C05453=1097.627,129.752,-63.111,176.753,16.480,152.163
C05454=1097.633,130.001,-63.131,176.756,16.481,152.163
C05455=1097.638,130.250,-63.150,176.760,16.481,152.162
C05456=1097.644,130.499,-63.171,176.762,16.481,152.162
C05457=1097.649,130.749,-63.190,176.765,16.482,152.161
C05458=1097.656,130.998,-63.210,176.768,16.482,152.161
C05459=1097.661,131.248,-63.229,176.771,16.482,152.160
C05460=1097.667,131.496,-63.249,176.774,16.482,152.159
C05461=1097.673,131.745,-63.270,176.777,16.482,152.159
C05462=1097.678,131.995,-63.289,176.780,16.482,152.158
C05463=1097.684,132.244,-63.309,176.783,16.483,152.158
C05464=1097.690,132.493,-63.329,176.785,16.483,152.157
C05465=1097.695,132.742,-63.349,176.789,16.483,152.157
C05466=1097.701,132.991,-63.369,176.792,16.484,152.156
C05467=1097.706,133.241,-63.389,176.794,16.484,152.156
C05468=1097.712,133.490,-63.409,176.798,16.484,152.155
C05469=1097.718,133.738,-63.429,176.801,16.484,152.155
C05470=1097.724,133.988,-63.449,176.803,16.485,152.154
C05471=1097.729,134.237,-63.468,176.806,16.485,152.154
C05472=1097.734,134.486,-63.489,176.810,16.485,152.153
C05473=1097.740,134.735,-63.509,176.812,16.485,152.152
C05474=1097.746,134.984,-63.528,176.815,16.485,152.152
C05475=1097.751,135.234,-63.549,176.819,16.486,152.151
C05476=1097.757,135.482,-63.569,176.821,16.486,152.151
C05477=1097.763,135.731,-63.589,176.824,16.486,152.150
C05478=1097.768,135.981,-63.608,176.828,16.486,152.150
C05479=1097.774,136.230,-63.629,176.830,16.486,152.149
C05480=1097.780,136.479,-63.649,176.833,16.487,152.149
C05481=1097.786,136.728,-63.669,176.836,16.487,152.148
C05482=1097.791,136.977,-63.689,176.839,16.487,152.147
C05483=1097.797,137.226,-63.709,176.842,16.488,152.147
C05484=1097.802,137.475,-63.729,176.845,16.488,152.146
C05485=1097.808,137.724,-63.749,176.848,16.488,152.146
C05486=1097.814,137.974,-63.770,176.851,16.488,152.145
C05487=1097.820,138.223,-63.790,176.854,16.489,152.145
C05488=1097.825,138.472,-63.811,176.857,16.488,152.144
C05489=1097.831,138.721,-63.831,176.860,16.489,152.143
C05490=1097.836,138.970,-63.850,176.863,16.489,152.143
C05491=1097.842,139.219,-63.870,176.866,16.489,152.142
C05492=1097.847,139.468,-63.891,176.869,16.489,152.142
C05493=1097.853,139.717,-63.911,176.872,16.490,152.141
C05494=1097.858,139.966,-63.931,176.875,16.489,152.141
C05495=1097.864,140.216,-63.952,176.878,16.490,152.140
C05496=1097.870,140.465,-63.972,176.881,16.490,152.139
C05497=1097.875,140.714,-63.993,176.884,16.490,152.139
C05498=1097.881,140.963,-64.013,176.887,16.490,152.138
C05499=1097.887,141.212,-64.033,176.890,16.490,152.138
C05500=1097.892,141.461,-64.054,176.893,16.490,152.137
C05501=1097.898,141.710,-64.074,176.896,16.491,152.137
C05502=1097.903,141.959,-64.094,176.899,16.491,152.136
C05503=1097.909,142.209,-64.115,176.902,16.491,152.135
C05504=1097.915,142.458,-64.135,176.905,16.491,152.135
C05505=1097.920,142.707,-64.156,176.908,16.492,152.134
C05506=1097.926,142.956,-64.176,176.912,16.492,152.134
C05507=1097.932,143.205,-64.196,176.914,16.492,152.133
C05508=1097.937,143.454,-64.217,176.917,16.492,152.133
C05509=1097.944,143.729,-64.240,176.921,16.492,152.132
C05510=1097.950,144.003,-64.262,176.924,16.492,152.131
C05511=1097.956,144.278,-64.286,176.928,16.492,152.130
C05512=1097.962,144.552,-64.308,176.931,16.493,152.130
C05513=1097.967,144.801,-64.329,176.934,16.493,152.129
C05514=1097.973,145.050,-64.348,176.937,16.493,152.129
C05515=1097.979,145.300,-64.369,176.940,16.493,152.128
C05516=1097.985,145.549,-64.390,176.943,16.493,152.128
C05517=1097.990,145.798,-64.410,176.946,16.493,152.127
C05518=1097.996,146.046,-64.431,176.949,16.493,152.126
C05519=1098.001,146.295,-64.452,176.953,16.494,152.126
C05520=1098.007,146.545,-64.473,176.955,16.493,152.125
C05521=1098.013,146.794,-64.493,176.959,16.494,152.125
C05522=1098.019,147.043,-64.513,176.962,16.494,152.124
C05523=1098.024,147.291,-64.534,176.964,16.494,152.123
C05524=1098.030,147.541,-64.555,176.968,16.494,152.123
C05525=1098.035,147.790,-64.576,176.971,16.494,152.122
C05526=1098.041,148.039,-64.596,176.974,16.494,152.122
C05527=1098.047,148.288,-64.617,176.977,16.494,152.121
C05528=1098.053,148.537,-64.638,176.980,16.494,152.120
C05529=1098.058,148.787,-64.659,176.984,16.495,152.120
C05530=1098.063,149.035,-64.680,176.986,16.494,152.119
C05531=1098.069,149.285,-64.701,176.989,16.495,152.119
C05532=1098.075,149.534,-64.721,176.993,16.495,152.118
C05533=1098.081,149.782,-64.742,176.995,16.495,152.117
C05534=1098.086,150.031,-64.763,176.999,16.495,152.117
C05535=1098.092,150.281,-64.783,177.002,16.495,152.116
C05536=1098.097,150.530,-64.805,177.005,16.495,152.115
C05537=1098.103,150.779,-64.825,177.008,16.495,152.115
C05538=1098.108,151.028,-64.846,177.012,16.495,152.114
C05539=1098.114,151.277,-64.868,177.015,16.496,152.114
C05540=1098.119,151.526,-64.888,177.017,16.495,152.113
C05541=1098.125,151.775,-64.909,177.021,16.496,152.112
C05542=1098.131,152.025,-64.930,177.024,16.496,152.112
C05543=1098.137,152.273,-64.951,177.027,16.495,152.111
C05544=1098.142,152.522,-64.971,177.030,16.495,152.110
C05545=1098.148,152.772,-64.992,177.033,16.496,152.110
C05546=1098.154,153.020,-65.014,177.037,16.496,152.109
C05547=1098.159,153.269,-65.034,177.039,16.496,152.109
C05548=1098.165,153.519,-65.056,177.043,16.496,152.108
C05549=1098.170,153.768,-65.076,177.046,16.496,152.107
C05550=1098.176,154.016,-65.098,177.049,16.496,152.107
C05551=1098.182,154.266,-65.119,177.052,16.496,152.106
C05552=1098.187,154.515,-65.140,177.055,16.496,152.105
C05553=1098.193,154.763,-65.161,177.059,16.496,152.105
C05554=1098.199,155.013,-65.182,177.061,16.496,152.104
C05555=1098.204,155.261,-65.203,177.065,16.496,152.104
C05556=1098.210,155.511,-65.224,177.068,16.497,152.103
C05557=1098.216,155.760,-65.246,177.071,16.496,152.102
C05558=1098.221,156.009,-65.266,177.074,16.496,152.102
C05559=1098.227,156.258,-65.288,177.078,16.496,152.101
C05560=1098.232,156.507,-65.310,177.081,16.497,152.100
C05561=1098.238,156.757,-65.330,177.084,16.496,152.100
C05562=1098.244,157.005,-65.352,177.087,16.497,152.099
C05563=1098.249,157.254,-65.373,177.090,16.496,152.098
C05564=1098.255,157.504,-65.394,177.094,16.497,152.098
C05565=1098.261,157.752,-65.415,177.096,16.496,152.097
C05566=1098.267,158.001,-65.437,177.100,16.497,152.097
C05567=1098.272,158.250,-65.457,177.103,16.497,152.096
C05568=1098.277,158.499,-65.479,177.106,16.496,152.095
C05569=1098.283,158.748,-65.501,177.109,16.496,152.095
C05570=1098.288,158.997,-65.521,177.112,16.497,152.094
C05571=1098.294,159.247,-65.543,177.116,16.497,152.093
C05572=1098.300,159.495,-65.564,177.118,16.497,152.093
C05573=1098.306,159.770,-65.588,177.122,16.497,152.092
C05574=1098.312,160.044,-65.611,177.126,16.496,152.091
C05575=1098.319,160.318,-65.635,177.129,16.496,152.091
C05576=1098.325,160.592,-65.659,177.133,16.496,152.090
C05577=1098.331,160.842,-65.680,177.136,16.496,152.089
C05578=1098.335,161.090,-65.701,177.139,16.497,152.089
C05579=1098.342,161.340,-65.723,177.143,16.497,152.088
C05580=1098.347,161.588,-65.744,177.146,16.497,152.087
C05581=1098.353,161.837,-65.766,177.149,16.496,152.087
C05582=1098.358,162.086,-65.788,177.152,16.497,152.086
C05583=1098.364,162.336,-65.809,177.156,16.497,152.085
C05584=1098.370,162.585,-65.830,177.158,16.497,152.085
C05585=1098.374,162.833,-65.852,177.162,16.497,152.084
C05586=1098.381,163.083,-65.874,177.165,16.497,152.083
C05587=1098.385,163.331,-65.895,177.169,16.497,152.083
C05588=1098.392,163.581,-65.917,177.171,16.496,152.082
C05589=1098.396,163.829,-65.939,177.175,16.497,152.081
C05590=1098.403,164.079,-65.961,177.178,16.497,152.081
C05591=1098.408,164.327,-65.982,177.181,16.497,152.080
C05592=1098.413,164.577,-66.004,177.184,16.497,152.079
C05593=1098.419,164.825,-66.025,177.188,16.497,152.079
C05594=1098.424,165.074,-66.047,177.191,16.497,152.078
C05595=1098.430,165.323,-66.069,177.195,16.497,152.077
C05596=1098.435,165.572,-66.091,177.198,16.497,152.077
C05597=1098.441,165.821,-66.112,177.201,16.497,152.076
C05598=1098.446,166.070,-66.134,177.204,16.497,152.075
C05599=1098.452,166.319,-66.156,177.207,16.497,152.075
C05600=1098.457,166.568,-66.178,177.211,16.497,152.074
C05601=1098.463,166.817,-66.199,177.214,16.496,152.073
C05602=1098.469,167.066,-66.221,177.217,16.497,152.073
C05603=1098.474,167.315,-66.243,177.221,16.497,152.072
C05604=1098.480,167.564,-66.264,177.224,16.497,152.071
C05605=1098.485,167.813,-66.286,177.227,16.497,152.071
C05606=1098.491,168.062,-66.308,177.230,16.497,152.070
C05607=1098.496,168.311,-66.330,177.234,16.497,152.069
C05608=1098.502,168.560,-66.351,177.237,16.497,152.069
C05609=1098.507,168.809,-66.374,177.240,16.496,152.068
C05610=1098.513,169.058,-66.396,177.243,16.496,152.067
C05611=1098.519,169.307,-66.418,177.247,16.496,152.067
C05612=1098.524,169.556,-66.440,177.250,16.497,152.066
C05613=1098.530,169.805,-66.461,177.254,16.497,152.065
C05614=1098.535,170.054,-66.483,177.256,16.496,152.065
C05615=1098.541,170.303,-66.506,177.260,16.496,152.064
C05616=1098.546,170.552,-66.527,177.263,16.496,152.063
C05617=1098.552,170.801,-66.549,177.267,16.496,152.063
C05618=1098.558,171.050,-66.571,177.269,16.496,152.062
C05619=1098.563,171.298,-66.593,177.273,16.496,152.061
C05620=1098.569,171.548,-66.616,177.276,16.496,152.061
C05621=1098.574,171.797,-66.638,177.280,16.496,152.060
C05622=1098.580,172.046,-66.659,177.283,16.496,152.059
C05623=1098.586,172.295,-66.682,177.286,16.495,152.059
C05624=1098.592,172.544,-66.704,177.290,16.495,152.058
C05625=1098.597,172.793,-66.726,177.293,16.495,152.057
C05626=1098.602,173.042,-66.748,177.297,16.495,152.056
C05627=1098.608,173.291,-66.770,177.299,16.495,152.056
C05628=1098.613,173.540,-66.792,177.303,16.495,152.055
C05629=1098.620,173.788,-66.814,177.306,16.495,152.054
C05630=1098.625,174.038,-66.837,177.310,16.495,152.054
C05631=1098.630,174.287,-66.858,177.313,16.495,152.053
C05632=1098.636,174.535,-66.881,177.316,16.495,152.052
C05633=1098.642,174.785,-66.903,177.320,16.495,152.052
C05634=1098.647,175.033,-66.926,177.323,16.494,152.051
C05635=1098.653,175.282,-66.947,177.327,16.494,152.050
C05636=1098.659,175.532,-66.969,177.329,16.494,152.049
C05637=1098.665,175.805,-66.994,177.334,16.494,152.049
C05638=1098.671,176.079,-67.019,177.338,16.494,152.048
C05639=1098.678,176.353,-67.043,177.341,16.494,152.047
C05640=1098.683,176.626,-67.068,177.345,16.493,152.046
C05641=1098.689,176.876,-67.089,177.349,16.493,152.045
C05642=1098.695,177.124,-67.112,177.351,16.493,152.045
C05643=1098.700,177.374,-67.135,177.355,16.493,152.044
C05644=1098.707,177.623,-67.157,177.358,16.493,152.043
C05645=1098.712,177.871,-67.180,177.362,16.493,152.043
C05646=1098.718,178.120,-67.202,177.365,16.492,152.042
C05647=1098.723,178.369,-67.225,177.368,16.492,152.041
C05648=1098.729,178.618,-67.246,177.372,16.492,152.040
C05649=1098.735,178.867,-67.269,177.375,16.492,152.040
C05650=1098.740,179.116,-67.291,177.379,16.492,152.039
C05651=1098.746,179.365,-67.314,177.382,16.491,152.038
C05652=1098.752,179.614,-67.336,177.385,16.491,152.038
C05653=1098.758,179.863,-67.359,177.389,16.491,152.037
C05654=1098.763,180.112,-67.382,177.392,16.491,152.036
C05655=1098.770,180.361,-67.404,177.396,16.491,152.035
C05656=1098.775,180.609,-67.426,177.399,16.490,152.035
C05657=1098.780,180.858,-67.449,177.402,16.490,152.034
C05658=1098.786,181.107,-67.472,177.406,16.490,152.033
C05659=1098.792,181.356,-67.493,177.410,16.490,152.032
C05660=1098.798,181.605,-67.516,177.413,16.490,152.032
C05661=1098.804,181.854,-67.539,177.416,16.490,152.031
C05662=1098.809,182.103,-67.562,177.420,16.489,152.030
C05663=1098.814,182.352,-67.584,177.423,16.489,152.029
C05664=1098.821,182.600,-67.606,177.427,16.489,152.029
C05665=1098.826,182.849,-67.629,177.430,16.489,152.028
C05666=1098.832,183.098,-67.652,177.433,16.489,152.027
C05667=1098.838,183.348,-67.675,177.437,16.488,152.026
C05668=1098.843,183.597,-67.698,177.440,16.488,152.026
C05669=1098.850,183.845,-67.720,177.444,16.488,152.025
C05670=1098.856,184.094,-67.743,177.448,16.488,152.024
C05671=1098.861,184.343,-67.766,177.451,16.487,152.023
C05672=1098.867,184.592,-67.789,177.454,16.487,152.023
C05673=1098.872,184.841,-67.811,177.458,16.487,152.022
C05674=1098.878,185.090,-67.834,177.461,16.487,152.021
C05675=1098.884,185.339,-67.857,177.465,16.487,152.020
C05676=1098.889,185.587,-67.879,177.469,16.487,152.020
C05677=1098.895,185.836,-67.902,177.471,16.486,152.019
C05678=1098.900,186.085,-67.925,177.475,16.486,152.018
C05679=1098.906,186.334,-67.948,177.478,16.486,152.017
C05680=1098.912,186.583,-67.971,177.482,16.486,152.017
C05681=1098.918,186.832,-67.994,177.486,16.486,152.016
C05682=1098.923,187.081,-68.017,177.489,16.486,152.015
C05683=1098.927,187.330,-68.040,177.492,16.485,152.015
C05684=1098.933,187.579,-68.062,177.496,16.485,152.014
C05685=1098.939,187.828,-68.085,177.499,16.485,152.013
C05686=1098.945,188.077,-68.108,177.503,16.485,152.012
C05687=1098.950,188.326,-68.131,177.506,16.485,152.012
C05688=1098.956,188.574,-68.154,177.510,16.485,152.011
C05689=1098.961,188.824,-68.178,177.513,16.484,152.010
C05690=1098.967,189.073,-68.201,177.516,16.484,152.009
C05691=1098.973,189.321,-68.224,177.520,16.484,152.009
C05692=1098.979,189.570,-68.247,177.523,16.484,152.008
C05693=1098.984,189.818,-68.270,177.527,16.484,152.007
C05694=1098.989,190.067,-68.293,177.531,16.483,152.006
C05695=1098.994,190.316,-68.316,177.534,16.483,152.006
C05696=1099.000,190.565,-68.339,177.537,16.483,152.005
C05697=1099.006,190.814,-68.362,177.541,16.483,152.004
C05698=1099.012,191.063,-68.385,177.545,16.482,152.003
C05699=1099.017,191.312,-68.409,177.548,16.482,152.003
C05700=1099.022,191.561,-68.432,177.552,16.482,152.002
C05701=1099.029,191.834,-68.458,177.555,16.482,152.001
C05702=1099.035,192.108,-68.483,177.559,16.482,152.000
C05703=1099.041,192.381,-68.509,177.563,16.482,151.999
C05704=1099.047,192.654,-68.535,177.567,16.481,151.998
C05705=1099.053,192.903,-68.557,177.570,16.481,151.998
C05706=1099.059,193.152,-68.580,177.574,16.481,151.997
C05707=1099.064,193.401,-68.604,177.578,16.481,151.996
C05708=1099.070,193.650,-68.627,177.581,16.481,151.995
C05709=1099.076,193.899,-68.651,177.584,16.480,151.995
C05710=1099.081,194.147,-68.674,177.588,16.480,151.994
C05711=1099.086,194.397,-68.697,177.591,16.480,151.993
C05712=1099.092,194.645,-68.721,177.595,16.479,151.992
C05713=1099.098,194.894,-68.744,177.599,16.479,151.992
C05714=1099.103,195.143,-68.767,177.602,16.479,151.991
C05715=1099.109,195.391,-68.791,177.606,16.479,151.990
C05716=1099.115,195.641,-68.814,177.609,16.478,151.989
C05717=1099.120,195.890,-68.838,177.613,16.478,151.988
C05718=1099.126,196.138,-68.861,177.616,16.478,151.988
C05719=1099.132,196.387,-68.884,177.620,16.478,151.987
C05720=1099.137,196.637,-68.908,177.623,16.477,151.986
C05721=1099.143,196.885,-68.932,177.627,16.478,151.985
C05722=1099.149,197.134,-68.954,177.631,16.477,151.984
C05723=1099.154,197.382,-68.979,177.634,16.477,151.984
C05724=1099.160,197.631,-69.002,177.637,16.476,151.983
C05725=1099.166,197.881,-69.025,177.641,16.476,151.982
C05726=1099.172,198.129,-69.049,177.645,16.476,151.981
C05727=1099.177,198.378,-69.072,177.648,16.476,151.981
C05728=1099.183,198.627,-69.096,177.652,16.475,151.980
C05729=1099.188,198.876,-69.119,177.656,16.475,151.979
C05730=1099.194,199.124,-69.143,177.660,16.475,151.978
C05731=1099.199,199.373,-69.167,177.662,16.474,151.977
C05732=1099.206,199.622,-69.191,177.666,16.474,151.977
C05733=1099.212,199.871,-69.214,177.670,16.474,151.976
C05734=1099.217,200.120,-69.238,177.674,16.473,151.975
C05735=1099.223,200.368,-69.261,177.677,16.473,151.974
C05736=1099.228,200.617,-69.285,177.681,16.473,151.973
C05737=1099.235,200.866,-69.309,177.684,16.473,151.973
C05738=1099.240,201.115,-69.332,177.688,16.473,151.972
C05739=1099.246,201.364,-69.356,177.691,16.472,151.971
C05740=1099.252,201.612,-69.380,177.695,16.472,151.970
C05741=1099.257,201.862,-69.404,177.699,16.471,151.969
C05742=1099.263,202.110,-69.427,177.702,16.471,151.969
C05743=1099.269,202.359,-69.452,177.706,16.471,151.968
C05744=1099.274,202.608,-69.475,177.710,16.470,151.967
C05745=1099.280,202.856,-69.499,177.713,16.470,151.966
C05746=1099.286,203.105,-69.523,177.717,16.470,151.965
C05747=1099.291,203.354,-69.547,177.720,16.469,151.965
C05748=1099.297,203.603,-69.570,177.724,16.469,151.964
C05749=1099.303,203.851,-69.594,177.727,16.469,151.963
C05750=1099.308,204.100,-69.618,177.731,16.469,151.962
C05751=1099.314,204.349,-69.642,177.735,16.469,151.962
C05752=1099.320,204.598,-69.666,177.739,16.468,151.961
C05753=1099.325,204.847,-69.691,177.742,16.468,151.960
C05754=1099.331,205.095,-69.713,177.746,16.468,151.959
C05755=1099.337,205.345,-69.738,177.750,16.468,151.958
C05756=1099.342,205.593,-69.762,177.753,16.467,151.957
C05757=1099.348,205.842,-69.786,177.756,16.466,151.957
C05758=1099.353,206.090,-69.810,177.760,16.466,151.956
C05759=1099.359,206.340,-69.834,177.764,16.466,151.955
C05760=1099.365,206.588,-69.858,177.767,16.466,151.954
C05761=1099.370,206.837,-69.882,177.771,16.466,151.953
C05762=1099.375,207.086,-69.906,177.775,16.465,151.953
C05763=1099.382,207.335,-69.930,177.778,16.465,151.952
C05764=1099.387,207.583,-69.955,177.782,16.465,151.951
C05765=1099.410,208.592,-70.052,177.824,16.478,151.946
C05766=1099.419,208.961,-70.089,177.829,16.479,151.945
C05767=1099.427,209.331,-70.125,177.833,16.480,151.944
C05768=1099.436,209.701,-70.161,177.839,16.480,151.943
C05769=1099.444,210.070,-70.197,177.844,16.482,151.942
C05770=1099.450,210.320,-70.222,177.847,16.482,151.941
C05771=1099.455,210.568,-70.246,177.851,16.482,151.941
C05772=1099.461,210.818,-70.271,177.855,16.483,151.940
C05773=1099.466,211.066,-70.296,177.858,16.484,151.940
C05774=1099.472,211.314,-70.320,177.861,16.484,151.939
C05775=1099.478,211.563,-70.344,177.864,16.485,151.939
C05776=1099.483,211.812,-70.369,177.868,16.485,151.938
C05777=1099.489,212.061,-70.393,177.872,16.486,151.938
C05778=1099.494,212.309,-70.418,177.875,16.486,151.937
C05779=1099.500,212.558,-70.443,177.878,16.487,151.936
C05780=1099.506,212.807,-70.467,177.882,16.487,151.936
C05781=1099.511,213.056,-70.491,177.885,16.488,151.935
C05782=1099.517,213.304,-70.517,177.889,16.489,151.935
C05783=1099.522,213.553,-70.541,177.892,16.489,151.934
C05784=1099.528,213.802,-70.566,177.895,16.490,151.934
C05785=1099.534,214.051,-70.590,177.899,16.490,151.933
C05786=1099.539,214.299,-70.615,177.903,16.492,151.932
C05787=1099.545,214.548,-70.639,177.906,16.492,151.932
C05788=1099.550,214.797,-70.664,177.909,16.493,151.931
C05789=1099.557,215.045,-70.689,177.912,16.493,151.931
C05790=1099.561,215.294,-70.714,177.916,16.494,151.930
C05791=1099.567,215.543,-70.739,177.920,16.494,151.930
C05792=1099.573,215.792,-70.764,177.923,16.495,151.929
C05793=1099.579,216.041,-70.788,177.926,16.495,151.928
C05794=1099.584,216.289,-70.813,177.930,16.496,151.928
C05795=1099.590,216.538,-70.838,177.934,16.497,151.927
C05796=1099.596,216.786,-70.863,177.937,16.497,151.927
C05797=1099.601,217.036,-70.888,177.940,16.498,151.926
C05798=1099.606,217.284,-70.913,177.943,16.498,151.926
C05799=1099.612,217.533,-70.938,177.947,16.499,151.925
C05800=1099.618,217.782,-70.962,177.951,16.500,151.925
C05801=1099.624,218.030,-70.987,177.954,16.500,151.924
C05802=1099.628,218.279,-71.012,177.957,16.501,151.923
C05803=1099.635,218.528,-71.037,177.961,16.502,151.923
C05804=1099.640,218.776,-71.062,177.965,16.502,151.922
C05805=1099.646,219.025,-71.087,177.968,16.503,151.922
C05806=1099.652,219.273,-71.112,177.971,16.503,151.921
C05807=1099.657,219.523,-71.137,177.975,16.504,151.921
C05808=1099.663,219.771,-71.162,177.978,16.505,151.920
C05809=1099.668,220.020,-71.187,177.982,16.505,151.919
C05810=1099.675,220.269,-71.212,177.985,16.506,151.919
C05811=1099.679,220.517,-71.238,177.989,16.507,151.918
C05812=1099.685,220.766,-71.262,177.992,16.507,151.918
C05813=1099.692,221.015,-71.288,177.995,16.508,151.917
C05814=1099.697,221.263,-71.313,177.999,16.508,151.917
C05815=1099.702,221.512,-71.338,178.003,16.509,151.916
C05816=1099.708,221.760,-71.363,178.006,16.510,151.915
C05817=1099.714,222.009,-71.388,178.009,16.510,151.915
C05818=1099.723,222.383,-71.426,178.014,16.511,151.914
C05819=1099.731,222.757,-71.464,178.020,16.512,151.913
C05820=1099.739,223.131,-71.501,178.025,16.514,151.913
C05821=1099.748,223.504,-71.540,178.030,16.514,151.912
C05822=1099.753,223.753,-71.565,178.033,16.515,151.911
C05823=1099.759,224.001,-71.590,178.037,16.516,151.910
C05824=1099.764,224.250,-71.615,178.041,16.517,151.910
C05825=1099.770,224.498,-71.641,178.044,16.517,151.909
C05826=1099.775,224.747,-71.667,178.047,16.518,151.909
C05827=1099.781,224.995,-71.692,178.051,16.519,151.908
C05828=1099.786,225.245,-71.717,178.054,16.519,151.908
C05829=1099.792,225.494,-71.742,178.058,16.520,151.907
C05830=1099.797,225.742,-71.768,178.062,16.521,151.907
C05831=1099.804,225.991,-71.793,178.065,16.521,151.906
C05832=1099.810,226.239,-71.819,178.068,16.522,151.906
C05833=1099.815,226.487,-71.844,178.071,16.522,151.905
C05834=1099.821,226.736,-71.869,178.075,16.524,151.904
C05835=1099.826,226.985,-71.895,178.079,16.524,151.904
C05836=1099.832,227.234,-71.921,178.082,16.525,151.903
C05837=1099.837,227.482,-71.946,178.086,16.526,151.903
C05838=1099.843,227.731,-71.972,178.089,16.526,151.902
C05839=1099.849,227.980,-71.998,178.093,16.526,151.902
C05840=1099.854,228.228,-72.023,178.097,16.527,151.901
C05841=1099.860,228.477,-72.048,178.100,16.528,151.900
C05842=1099.866,228.726,-72.074,178.103,16.528,151.900
C05843=1099.872,228.974,-72.100,178.107,16.530,151.899
C05844=1099.877,229.223,-72.125,178.110,16.530,151.899
C05845=1099.883,229.471,-72.151,178.114,16.531,151.898
C05846=1099.888,229.720,-72.177,178.117,16.531,151.898
C05847=1099.895,229.969,-72.202,178.121,16.532,151.897
C05848=1099.900,230.218,-72.228,178.124,16.533,151.897
C05849=1099.905,230.466,-72.253,178.127,16.533,151.896
C05850=1099.911,230.715,-72.279,178.131,16.534,151.896
C05851=1099.917,230.963,-72.305,178.135,16.535,151.895
C05852=1099.922,231.212,-72.331,178.138,16.536,151.894
C05853=1099.928,231.460,-72.356,178.142,16.537,151.894
C05854=1099.933,231.709,-72.382,178.145,16.537,151.893
C05855=1099.939,231.958,-72.408,178.148,16.538,151.893
C05856=1099.944,232.207,-72.434,178.152,16.539,151.892
C05857=1099.951,232.455,-72.460,178.156,16.539,151.892
C05858=1099.956,232.703,-72.486,178.159,16.540,151.891
C05859=1099.961,232.952,-72.512,178.163,16.541,151.891
C05860=1099.967,233.201,-72.537,178.166,16.542,151.890
C05861=1099.973,233.449,-72.564,178.169,16.542,151.890
C05862=1099.979,233.698,-72.590,178.173,16.543,151.889
C05863=1099.984,233.947,-72.615,178.176,16.544,151.888
C05864=1099.990,234.195,-72.641,178.180,16.544,151.888
C05865=1099.995,234.444,-72.667,178.184,16.545,151.887
C05866=1100.001,234.693,-72.693,178.187,16.546,151.887
C05867=1100.007,234.941,-72.720,178.191,16.547,151.886
C05868=1100.012,235.190,-72.746,178.194,16.548,151.886
C05869=1100.018,235.439,-72.772,178.197,16.549,151.885
C05870=1100.025,235.803,-72.810,178.203,16.549,151.884
C05871=1100.034,236.169,-72.848,178.208,16.551,151.884
C05872=1100.042,236.534,-72.887,178.213,16.552,151.883
C05873=1100.050,236.899,-72.925,178.218,16.553,151.882
C05874=1100.056,237.148,-72.951,178.221,16.554,151.882
C05875=1100.062,237.396,-72.977,178.225,16.555,151.881
C05876=1100.068,237.645,-73.003,178.228,16.556,151.881
C05877=1100.074,237.893,-73.030,178.232,16.557,151.880
C05878=1100.079,238.142,-73.056,178.236,16.557,151.880
C05879=1100.084,238.390,-73.082,178.239,16.558,151.879
C05880=1100.090,238.639,-73.108,178.243,16.559,151.878
C05881=1100.096,238.887,-73.134,178.246,16.559,151.878
C05882=1100.101,239.136,-73.160,178.249,16.560,151.877
C05883=1100.107,239.384,-73.187,178.253,16.561,151.877
C05884=1100.112,239.633,-73.213,178.256,16.562,151.876
C05885=1100.118,239.882,-73.240,178.260,16.563,151.876
C05886=1100.124,240.130,-73.266,178.264,16.563,151.875
C05887=1100.129,240.379,-73.292,178.267,16.564,151.875
C05888=1100.135,240.628,-73.319,178.271,16.565,151.874
C05889=1100.141,240.877,-73.345,178.274,16.566,151.874
C05890=1100.146,241.125,-73.371,178.277,16.567,151.873
C05891=1100.152,241.373,-73.398,178.281,16.568,151.873
C05892=1100.158,241.622,-73.425,178.284,16.568,151.872
C05893=1100.163,241.871,-73.451,178.288,16.569,151.872
C05894=1100.169,242.119,-73.477,178.292,16.570,151.871
C05895=1100.175,242.367,-73.504,178.295,16.570,151.870
C05896=1100.180,242.616,-73.530,178.299,16.572,151.870
C05897=1100.186,242.865,-73.557,178.302,16.572,151.869
C05898=1100.192,243.113,-73.583,178.306,16.573,151.869
C05899=1100.198,243.361,-73.610,178.309,16.574,151.868
C05900=1100.203,243.610,-73.636,178.312,16.575,151.868
C05901=1100.209,243.859,-73.662,178.316,16.576,151.867
C05902=1100.214,244.107,-73.690,178.319,16.576,151.867
C05903=1100.220,244.356,-73.716,178.323,16.578,151.866
C05904=1100.225,244.604,-73.743,178.327,16.578,151.866
C05905=1100.231,244.852,-73.770,178.331,16.579,151.865
C05906=1100.237,245.101,-73.796,178.334,16.580,151.865
C05907=1100.242,245.350,-73.823,178.337,16.581,151.864
C05908=1100.248,245.598,-73.849,178.341,16.582,151.864
C05909=1100.253,245.847,-73.876,178.344,16.583,151.863
C05910=1100.259,246.095,-73.903,178.348,16.584,151.863
C05911=1100.265,246.344,-73.930,178.351,16.585,151.862
C05912=1100.271,246.593,-73.957,178.355,16.586,151.862
C05913=1100.276,246.841,-73.984,178.358,16.586,151.861
C05914=1100.282,247.090,-74.010,178.361,16.587,151.861
C05915=1100.288,247.338,-74.037,178.365,16.588,151.860
C05916=1100.293,247.587,-74.064,178.369,16.589,151.860
C05917=1100.299,247.835,-74.091,178.372,16.590,151.859
C05918=1100.304,248.083,-74.117,178.376,16.591,151.859
C05919=1100.309,248.332,-74.145,178.380,16.592,151.858
C05920=1100.315,248.580,-74.171,178.383,16.593,151.858
C05921=1100.320,248.829,-74.199,178.387,16.594,151.857
C05922=1100.328,249.187,-74.237,178.391,16.595,151.857
C05923=1100.337,249.545,-74.276,178.396,16.596,151.856
C05924=1100.344,249.904,-74.315,178.401,16.597,151.855
C05925=1100.353,250.263,-74.354,178.406,16.599,151.854
C05926=1100.358,250.511,-74.382,178.410,16.600,151.854
C05927=1100.364,250.760,-74.408,178.413,16.601,151.853
C05928=1100.370,251.008,-74.435,178.417,16.602,151.853
C05929=1100.375,251.256,-74.463,178.420,16.603,151.852
C05930=1100.381,251.504,-74.489,178.424,16.604,151.852
C05931=1100.386,251.753,-74.517,178.427,16.605,151.851
C05932=1100.392,252.001,-74.543,178.431,16.606,151.851
C05933=1100.397,252.251,-74.571,178.434,16.607,151.850
C05934=1100.403,252.498,-74.598,178.438,16.608,151.850
C05935=1100.408,252.747,-74.626,178.441,16.609,151.849
C05936=1100.414,252.996,-74.652,178.445,16.610,151.849
C05937=1100.419,253.244,-74.679,178.449,16.610,151.848
C05938=1100.426,253.493,-74.707,178.452,16.612,151.848
C05939=1100.431,253.741,-74.734,178.456,16.613,151.847
C05940=1100.437,253.990,-74.761,178.459,16.613,151.847
C05941=1100.442,254.238,-74.789,178.462,16.615,151.847
C05942=1100.448,254.486,-74.816,178.466,16.615,151.846
C05943=1100.454,254.735,-74.844,178.470,16.616,151.845
C05944=1100.459,254.983,-74.871,178.473,16.617,151.845
C05945=1100.464,255.232,-74.898,178.477,16.619,151.845
C05946=1100.471,255.480,-74.925,178.480,16.619,151.844
C05947=1100.476,255.729,-74.953,178.484,16.620,151.843
C05948=1100.482,255.977,-74.981,178.487,16.621,151.843
C05949=1100.487,256.225,-75.008,178.491,16.622,151.843
C05950=1100.492,256.474,-75.035,178.494,16.623,151.842
C05951=1100.499,256.722,-75.062,178.498,16.624,151.841
C05952=1100.504,256.971,-75.090,178.501,16.625,151.841
C05953=1100.510,257.219,-75.117,178.505,16.626,151.841
C05954=1100.516,257.468,-75.145,178.508,16.627,151.840
C05955=1100.521,257.716,-75.173,178.512,16.629,151.840
C05956=1100.527,257.964,-75.200,178.515,16.629,151.839
C05957=1100.532,258.213,-75.227,178.519,16.630,151.839
C05958=1100.538,258.461,-75.256,178.522,16.631,151.838
C05959=1100.544,258.710,-75.282,178.526,16.632,151.838
C05960=1100.549,258.958,-75.310,178.529,16.633,151.837
C05961=1100.556,259.206,-75.338,178.533,16.634,151.837
C05962=1100.561,259.455,-75.365,178.536,16.635,151.836
C05963=1100.566,259.703,-75.393,178.540,16.636,151.836
C05964=1100.573,259.952,-75.420,178.543,16.637,151.835
C05965=1100.578,260.200,-75.448,178.547,16.638,151.835
C05966=1100.584,260.449,-75.476,178.550,16.639,151.834
C05967=1100.590,260.697,-75.504,178.554,16.640,151.834
C05968=1100.595,260.945,-75.531,178.558,16.641,151.833
C05969=1100.601,261.194,-75.559,178.561,16.642,151.833
C05970=1100.607,261.442,-75.587,178.565,16.643,151.832
C05971=1100.613,261.691,-75.614,178.569,16.644,151.832
C05972=1100.618,261.939,-75.642,178.571,16.645,151.831
C05973=1100.623,262.187,-75.670,178.575,16.646,151.831
C05974=1100.633,262.543,-75.710,178.581,16.648,151.830
C05975=1100.640,262.898,-75.749,178.586,16.649,151.829
C05976=1100.649,263.254,-75.790,178.591,16.650,151.829
C05977=1100.657,263.609,-75.829,178.596,16.652,151.828
C05978=1100.663,263.858,-75.858,178.599,16.653,151.828
C05979=1100.669,264.105,-75.885,178.603,16.654,151.827
C05980=1100.675,264.354,-75.913,178.607,16.655,151.827
C05981=1100.680,264.602,-75.941,178.610,16.656,151.826
C05982=1100.686,264.852,-75.969,178.614,16.657,151.826
C05983=1100.691,265.100,-75.997,178.617,16.658,151.825
C05984=1100.697,265.348,-76.025,178.621,16.659,151.825
C05985=1100.702,265.596,-76.053,178.623,16.660,151.824
C05986=1100.708,265.844,-76.081,178.627,16.662,151.824
C05987=1100.713,266.093,-76.109,178.631,16.663,151.823
C05988=1100.719,266.341,-76.137,178.634,16.664,151.823
C05989=1100.725,266.590,-76.166,178.638,16.665,151.823
C05990=1100.730,266.838,-76.194,178.641,16.666,151.822
C05991=1100.736,267.087,-76.222,178.645,16.668,151.822
C05992=1100.741,267.335,-76.250,178.648,16.668,151.821
C05993=1100.747,267.584,-76.278,178.652,16.670,151.821
C05994=1100.753,267.832,-76.306,178.656,16.671,151.820
C05995=1100.759,268.080,-76.335,178.659,16.672,151.820
C05996=1100.764,268.328,-76.363,178.663,16.673,151.819
C05997=1100.770,268.577,-76.392,178.666,16.674,151.819
C05998=1100.776,268.825,-76.420,178.670,16.675,151.818
C05999=1100.781,269.073,-76.448,178.673,16.676,151.818
C06000=1100.787,269.321,-76.476,178.677,16.678,151.818
C06001=1100.793,269.570,-76.504,178.680,16.679,151.817
C06002=1100.798,269.818,-76.533,178.684,16.680,151.817
C06003=1100.804,270.066,-76.561,178.687,16.681,151.816
C06004=1100.810,270.314,-76.589,178.691,16.682,151.816
C06005=1100.816,270.563,-76.617,178.694,16.684,151.815
C06006=1100.821,270.811,-76.645,178.697,16.684,151.815
C06007=1100.827,271.059,-76.674,178.701,16.686,151.814
C06008=1100.833,271.307,-76.702,178.705,16.687,151.814
C06009=1100.838,271.556,-76.731,178.708,16.688,151.814
C06010=1100.843,271.804,-76.760,178.712,16.690,151.813
C06011=1100.849,272.053,-76.788,178.715,16.690,151.813
C06012=1100.855,272.301,-76.817,178.719,16.692,151.812
C06013=1100.861,272.549,-76.845,178.723,16.693,151.812
C06014=1100.867,272.798,-76.874,178.726,16.694,151.811
C06015=1100.872,273.046,-76.902,178.729,16.696,151.811
C06016=1100.878,273.294,-76.931,178.733,16.696,151.811
C06017=1100.884,273.543,-76.960,178.736,16.698,151.810
C06018=1100.889,273.791,-76.988,178.740,16.699,151.810
C06019=1100.895,274.039,-77.017,178.743,16.700,151.809
C06020=1100.900,274.287,-77.045,178.747,16.702,151.809
C06021=1100.906,274.535,-77.074,178.750,16.702,151.808
C06022=1100.912,274.784,-77.102,178.754,16.704,151.808
C06023=1100.917,275.032,-77.132,178.757,16.705,151.808
C06024=1100.923,275.281,-77.160,178.761,16.706,151.807
C06025=1100.929,275.528,-77.189,178.764,16.708,151.807
C06026=1100.936,275.887,-77.230,178.769,16.710,151.806
C06027=1100.944,276.245,-77.271,178.774,16.711,151.806
C06028=1100.953,276.603,-77.313,178.780,16.713,151.805
C06029=1100.961,276.962,-77.354,178.785,16.715,151.804
C06030=1100.966,277.210,-77.384,178.788,16.716,151.804
C06031=1100.972,277.458,-77.412,178.791,16.717,151.804
C06032=1100.979,277.707,-77.441,178.795,16.719,151.803
C06033=1100.983,277.954,-77.470,178.798,16.720,151.803
C06034=1100.989,278.203,-77.499,178.802,16.721,151.802
C06035=1100.995,278.452,-77.528,178.806,16.723,151.802
C06036=1101.001,278.699,-77.557,178.809,16.724,151.802
C06037=1101.007,278.948,-77.585,178.812,16.725,151.801
C06038=1101.012,279.196,-77.615,178.816,16.727,151.801
C06039=1101.018,279.444,-77.644,178.819,16.728,151.800
C06040=1101.023,279.692,-77.673,178.823,16.729,151.800
C06041=1101.029,279.941,-77.702,178.826,16.730,151.800
C06042=1101.034,280.188,-77.731,178.830,16.732,151.799
C06043=1101.040,280.437,-77.760,178.834,16.733,151.799
C06044=1101.047,280.685,-77.789,178.837,16.734,151.798
C06045=1101.052,280.934,-77.818,178.840,16.736,151.798
C06046=1101.057,281.181,-77.847,178.844,16.737,151.797
C06047=1101.063,281.430,-77.876,178.847,16.738,151.797
C06048=1101.068,281.678,-77.906,178.851,16.740,151.797
C06049=1101.075,281.926,-77.935,178.855,16.741,151.796
C06050=1101.079,282.175,-77.963,178.858,16.742,151.796
C06051=1101.086,282.423,-77.992,178.861,16.744,151.796
C06052=1101.091,282.671,-78.022,178.865,16.745,151.795
C06053=1101.097,282.920,-78.052,178.868,16.746,151.795
C06054=1101.102,283.167,-78.080,178.872,16.748,151.794
C06055=1101.108,283.416,-78.110,178.876,16.749,151.794
C06056=1101.114,283.664,-78.139,178.878,16.750,151.794
C06057=1101.119,283.912,-78.169,178.882,16.752,151.793
C06058=1101.124,284.160,-78.198,178.886,16.754,151.793
C06059=1101.131,284.408,-78.227,178.890,16.755,151.793
C06060=1101.136,284.656,-78.257,178.892,16.756,151.792
C06061=1101.142,284.905,-78.286,178.896,16.758,151.792
C06062=1101.147,285.152,-78.315,178.900,16.760,151.791
C06063=1101.153,285.401,-78.345,178.903,16.760,151.791
C06064=1101.158,285.649,-78.374,178.907,16.762,151.791
C06065=1101.165,285.897,-78.403,178.910,16.764,151.790
C06066=1101.170,286.146,-78.433,178.913,16.765,151.790
C06067=1101.176,286.394,-78.463,178.917,16.766,151.789
C06068=1101.181,286.642,-78.491,178.921,16.768,151.789
C06069=1101.187,286.890,-78.521,178.924,16.769,151.789
C06070=1101.193,287.138,-78.551,178.927,16.770,151.788
C06071=1101.198,287.386,-78.581,178.931,16.772,151.788
C06072=1101.204,287.634,-78.610,178.935,16.774,151.788
C06073=1101.210,287.883,-78.640,178.938,16.775,151.787
C06074=1101.215,288.131,-78.669,178.941,16.776,151.787
C06075=1101.221,288.379,-78.698,178.945,16.778,151.787
C06076=1101.227,288.627,-78.728,178.948,16.779,151.786
C06077=1101.232,288.875,-78.758,178.952,16.781,151.786
C06078=1101.241,289.243,-78.802,178.957,16.783,151.785
C06079=1101.249,289.610,-78.846,178.962,16.785,151.785
C06080=1101.258,289.978,-78.890,178.968,16.787,151.784
C06081=1101.266,290.345,-78.934,178.972,16.789,151.784
C06082=1101.272,290.593,-78.964,178.976,16.791,151.783
C06083=1101.277,290.842,-78.993,178.980,16.793,151.783
C06084=1101.283,291.090,-79.024,178.983,16.794,151.783
C06085=1101.289,291.338,-79.053,178.986,16.795,151.782
C06086=1101.295,291.586,-79.082,178.990,16.797,151.782
C06087=1101.300,291.834,-79.113,178.994,16.799,151.782
C06088=1101.306,292.083,-79.142,178.996,16.800,151.781
C06089=1101.312,292.330,-79.173,179.000,16.802,151.781
C06090=1101.317,292.579,-79.202,179.004,16.803,151.781
C06091=1101.323,292.827,-79.232,179.007,16.805,151.780
C06092=1101.329,293.075,-79.262,179.010,16.806,151.780
C06093=1101.334,293.323,-79.292,179.014,16.808,151.780
C06094=1101.340,293.571,-79.322,179.018,16.809,151.779
C06095=1101.345,293.819,-79.351,179.021,16.811,151.779
C06096=1101.351,294.067,-79.382,179.024,16.812,151.779
C06097=1101.356,294.315,-79.411,179.028,16.814,151.778
C06098=1101.362,294.563,-79.442,179.031,16.816,151.778
C06099=1101.368,294.811,-79.472,179.035,16.817,151.778
C06100=1101.373,295.059,-79.502,179.038,16.818,151.777
C06101=1101.379,295.307,-79.532,179.042,16.820,151.777
C06102=1101.385,295.556,-79.562,179.045,16.822,151.777
C06103=1101.390,295.803,-79.592,179.049,16.824,151.776
C06104=1101.396,296.051,-79.622,179.053,16.825,151.776
C06105=1101.402,296.300,-79.652,179.056,16.826,151.776
C06106=1101.408,296.548,-79.683,179.059,16.828,151.775
C06107=1101.414,296.796,-79.713,179.063,16.830,151.775
C06108=1101.420,297.045,-79.743,179.066,16.832,151.775
C06109=1101.425,297.293,-79.774,179.069,16.833,151.774
C06110=1101.430,297.540,-79.804,179.073,16.835,151.774
C06111=1101.436,297.788,-79.834,179.076,16.836,151.774
C06112=1101.442,298.037,-79.864,179.080,16.838,151.773
C06113=1101.448,298.285,-79.894,179.083,16.840,151.773
C06114=1101.453,298.532,-79.925,179.086,16.841,151.773
C06115=1101.458,298.781,-79.956,179.090,16.843,151.773
C06116=1101.464,299.029,-79.985,179.093,16.845,151.772
C06117=1101.470,299.277,-80.016,179.097,16.847,151.772
C06118=1101.475,299.525,-80.047,179.101,16.849,151.772
C06119=1101.481,299.773,-80.077,179.104,16.850,151.771
C06120=1101.487,300.021,-80.107,179.107,16.852,151.771
C06121=1101.492,300.268,-80.138,179.111,16.853,151.771
C06122=1101.497,300.517,-80.168,179.114,16.855,151.771
C06123=1101.503,300.765,-80.198,179.118,16.857,151.770
C06124=1101.509,301.013,-80.229,179.121,16.859,151.770
C06125=1101.514,301.261,-80.260,179.125,16.861,151.770
C06126=1101.520,301.509,-80.290,179.127,16.862,151.770
C06127=1101.525,301.757,-80.321,179.131,16.864,151.769
C06128=1101.531,302.005,-80.351,179.134,16.866,151.769
C06129=1101.537,302.253,-80.382,179.138,16.868,151.769
C06130=1101.545,302.634,-80.429,179.143,16.871,151.768
C06131=1101.554,303.015,-80.476,179.149,16.873,151.768
C06132=1101.562,303.397,-80.523,179.154,16.876,151.767
C06133=1101.571,303.779,-80.571,179.159,16.879,151.767
C06134=1101.576,304.026,-80.601,179.163,16.881,151.767
C06135=1101.582,304.275,-80.632,179.166,16.882,151.766
C06136=1101.588,304.523,-80.663,179.169,16.884,151.766
C06137=1101.594,304.770,-80.694,179.173,16.886,151.766
C06138=1101.599,305.018,-80.725,179.176,16.888,151.766
C06139=1101.605,305.266,-80.755,179.180,16.890,151.766
C06140=1101.610,305.514,-80.786,179.183,16.891,151.765
C06141=1101.616,305.763,-80.817,179.187,16.894,151.765
C06142=1101.621,306.011,-80.847,179.190,16.895,151.765
C06143=1101.628,306.258,-80.879,179.193,16.897,151.764
C06144=1101.633,306.506,-80.909,179.196,16.899,151.764
C06145=1101.638,306.754,-80.940,179.200,16.900,151.764
C06146=1101.644,307.003,-80.971,179.204,16.902,151.764
C06147=1101.650,307.250,-81.002,179.207,16.904,151.763
C06148=1101.655,307.498,-81.033,179.211,16.906,151.763
C06149=1101.661,307.746,-81.064,179.214,16.908,151.763
C06150=1101.667,307.995,-81.095,179.218,16.910,151.763
C06151=1101.673,308.242,-81.126,179.220,16.911,151.762
C06152=1101.678,308.490,-81.157,179.224,16.913,151.762
C06153=1101.684,308.738,-81.188,179.227,16.915,151.762
C06154=1101.690,308.986,-81.219,179.231,16.917,151.762
C06155=1101.696,309.234,-81.250,179.234,16.919,151.762
C06156=1101.701,309.482,-81.281,179.238,16.921,151.761
C06157=1101.707,309.730,-81.312,179.241,16.923,151.761
C06158=1101.713,309.978,-81.343,179.245,16.925,151.761
C06159=1101.718,310.226,-81.375,179.248,16.927,151.761
C06160=1101.724,310.474,-81.405,179.252,16.929,151.760
C06161=1101.730,310.722,-81.437,179.254,16.930,151.760
C06162=1101.736,310.970,-81.467,179.258,16.932,151.760
C06163=1101.742,311.218,-81.499,179.262,16.934,151.760
C06164=1101.747,311.466,-81.530,179.265,16.936,151.759
C06165=1101.753,311.713,-81.561,179.268,16.938,151.759
C06166=1101.758,311.962,-81.593,179.272,16.940,151.759
C06167=1101.764,312.210,-81.624,179.275,16.942,151.759
C06168=1101.770,312.458,-81.655,179.279,16.944,151.758
C06169=1101.776,312.706,-81.687,179.282,16.946,151.758
C06170=1101.782,312.953,-81.718,179.286,16.948,151.758
C06171=1101.787,313.202,-81.749,179.288,16.950,151.758
C06172=1101.793,313.449,-81.781,179.292,16.951,151.758
C06173=1101.800,313.697,-81.812,179.295,16.953,151.757
C06174=1101.805,313.945,-81.843,179.299,16.955,151.757
C06175=1101.811,314.194,-81.875,179.302,16.958,151.757
C06176=1101.816,314.441,-81.907,179.306,16.960,151.757
C06177=1101.822,314.690,-81.937,179.309,16.961,151.756
C06178=1101.828,314.937,-81.969,179.313,16.963,151.756
C06179=1101.834,315.185,-82.001,179.316,16.965,151.756
C06180=1101.840,315.433,-82.032,179.319,16.968,151.756
C06181=1101.845,315.681,-82.063,179.323,16.970,151.756
C06182=1101.854,316.065,-82.113,179.328,16.973,151.755
C06183=1101.862,316.449,-82.161,179.333,16.976,151.755
C06184=1101.870,316.834,-82.211,179.338,16.979,151.755
C06185=1101.879,317.217,-82.260,179.343,16.983,151.755
C06186=1101.884,317.465,-82.291,179.346,16.985,151.755
C06187=1101.890,317.713,-82.324,179.350,16.987,151.754
C06188=1101.896,317.960,-82.355,179.353,16.989,151.754
C06189=1101.901,318.209,-82.386,179.356,16.991,151.754
C06190=1101.907,318.457,-82.418,179.360,16.993,151.754
C06191=1101.913,318.705,-82.450,179.363,16.995,151.754
C06192=1101.918,318.952,-82.482,179.366,16.998,151.754
C06193=1101.924,319.201,-82.514,179.370,17.000,151.754
C06194=1101.929,319.448,-82.546,179.373,17.002,151.753
C06195=1101.935,319.696,-82.578,179.376,17.004,151.753
C06196=1101.941,319.944,-82.609,179.380,17.006,151.753
C06197=1101.947,320.192,-82.641,179.383,17.009,151.753
C06198=1101.952,320.440,-82.673,179.386,17.011,151.753
C06199=1101.958,320.688,-82.705,179.390,17.013,151.753
C06200=1101.964,320.935,-82.737,179.393,17.016,151.753
C06201=1101.969,321.184,-82.769,179.396,17.018,151.752
C06202=1101.974,321.431,-82.801,179.400,17.020,151.752
C06203=1101.980,321.680,-82.833,179.403,17.022,151.752
C06204=1101.986,321.927,-82.865,179.406,17.024,151.752
C06205=1101.992,322.175,-82.897,179.410,17.026,151.752
C06206=1101.997,322.423,-82.928,179.413,17.029,151.752
C06207=1102.003,322.671,-82.960,179.416,17.031,151.752
C06208=1102.008,322.918,-82.993,179.419,17.033,151.751
C06209=1102.014,323.166,-83.025,179.423,17.036,151.751
C06210=1102.020,323.415,-83.057,179.426,17.038,151.751
C06211=1102.025,323.662,-83.089,179.429,17.040,151.751
C06212=1102.031,323.910,-83.121,179.432,17.042,151.751
C06213=1102.037,324.158,-83.153,179.436,17.044,151.751
C06214=1102.042,324.406,-83.186,179.440,17.047,151.751
C06215=1102.048,324.654,-83.218,179.443,17.050,151.751
C06216=1102.054,324.901,-83.250,179.447,17.052,151.750
C06217=1102.060,325.150,-83.282,179.450,17.054,151.750
C06218=1102.065,325.398,-83.315,179.453,17.056,151.750
C06219=1102.070,325.645,-83.347,179.456,17.059,151.750
C06220=1102.076,325.893,-83.379,179.460,17.061,151.750
C06221=1102.083,326.141,-83.411,179.463,17.063,151.750
C06222=1102.088,326.388,-83.443,179.466,17.065,151.750
C06223=1102.093,326.637,-83.476,179.469,17.068,151.750
C06224=1102.100,326.885,-83.508,179.473,17.070,151.750
C06225=1102.105,327.132,-83.540,179.476,17.072,151.750
C06226=1102.110,327.381,-83.573,179.479,17.075,151.749
C06227=1102.117,327.628,-83.606,179.482,17.077,151.749
C06228=1102.123,327.876,-83.638,179.486,17.079,151.749
C06229=1102.128,328.123,-83.670,179.489,17.082,151.749
C06230=1102.134,328.372,-83.703,179.492,17.084,151.749
C06231=1102.140,328.619,-83.735,179.496,17.087,151.749
C06232=1102.146,328.868,-83.767,179.499,17.089,151.749
C06233=1102.151,329.115,-83.800,179.503,17.091,151.749
C06234=1102.160,329.492,-83.849,179.507,17.095,151.749
C06235=1102.169,329.869,-83.899,179.512,17.099,151.749
C06236=1102.177,330.246,-83.948,179.517,17.102,151.748
C06237=1102.186,330.623,-83.998,179.523,17.106,151.748
C06238=1102.192,330.871,-84.031,179.526,17.109,151.748
C06239=1102.198,331.119,-84.063,179.529,17.111,151.748
C06240=1102.204,331.367,-84.096,179.532,17.113,151.748
C06241=1102.209,331.614,-84.129,179.535,17.116,151.748
C06242=1102.215,331.862,-84.161,179.539,17.118,151.748
C06243=1102.221,332.110,-84.194,179.542,17.120,151.748
C06244=1102.227,332.357,-84.227,179.545,17.123,151.748
C06245=1102.232,332.606,-84.259,179.549,17.126,151.748
C06246=1102.239,332.853,-84.292,179.552,17.129,151.748
C06247=1102.244,333.101,-84.325,179.555,17.131,151.748
C06248=1102.249,333.349,-84.358,179.558,17.134,151.748
C06249=1102.255,333.597,-84.390,179.562,17.136,151.748
C06250=1102.261,333.845,-84.424,179.565,17.138,151.748
C06251=1102.266,334.093,-84.457,179.568,17.141,151.748
C06252=1102.272,334.339,-84.490,179.572,17.144,151.747
C06253=1102.277,334.588,-84.522,179.575,17.146,151.747
C06254=1102.284,334.836,-84.555,179.578,17.149,151.747
C06255=1102.289,335.083,-84.588,179.581,17.151,151.747
C06256=1102.295,335.331,-84.622,179.584,17.154,151.747
C06257=1102.301,335.579,-84.654,179.587,17.157,151.748
C06258=1102.306,335.826,-84.687,179.591,17.160,151.748
C06259=1102.311,336.074,-84.721,179.594,17.162,151.748
C06260=1102.318,336.322,-84.753,179.597,17.165,151.747
C06261=1102.323,336.570,-84.786,179.600,17.167,151.747
C06262=1102.329,336.818,-84.819,179.603,17.170,151.747
C06263=1102.335,337.066,-84.852,179.607,17.173,151.747
C06264=1102.340,337.314,-84.885,179.610,17.176,151.747
C06265=1102.346,337.562,-84.919,179.613,17.178,151.747
C06266=1102.352,337.809,-84.952,179.617,17.181,151.747
C06267=1102.357,338.056,-84.984,179.619,17.183,151.748
C06268=1102.363,338.304,-85.018,179.623,17.187,151.747
C06269=1102.369,338.551,-85.052,179.626,17.189,151.747
C06270=1102.375,338.799,-85.085,179.630,17.192,151.747
C06271=1102.380,339.047,-85.118,179.633,17.194,151.747
C06272=1102.386,339.295,-85.151,179.635,17.197,151.748
C06273=1102.392,339.543,-85.185,179.639,17.200,151.748
C06274=1102.397,339.791,-85.218,179.642,17.203,151.748
C06275=1102.403,340.039,-85.251,179.645,17.206,151.748
C06276=1102.408,340.287,-85.285,179.648,17.208,151.748
C06277=1102.415,340.534,-85.317,179.652,17.212,151.748
C06278=1102.420,340.781,-85.351,179.655,17.214,151.748
C06279=1102.426,341.029,-85.385,179.658,17.217,151.748
C06280=1102.432,341.277,-85.418,179.661,17.220,151.748
C06281=1102.437,341.525,-85.451,179.665,17.223,151.748
C06282=1102.442,341.772,-85.485,179.668,17.226,151.748
C06283=1102.448,342.020,-85.518,179.671,17.228,151.748
C06284=1102.453,342.267,-85.552,179.674,17.231,151.748
C06285=1102.459,342.515,-85.585,179.678,17.234,151.748
C06286=1102.468,342.886,-85.635,179.682,17.238,151.748
C06287=1102.476,343.257,-85.686,179.687,17.243,151.748
C06288=1102.485,343.628,-85.736,179.692,17.247,151.748
C06289=1102.494,343.998,-85.786,179.696,17.251,151.749
C06290=1102.499,344.246,-85.819,179.700,17.255,151.749
C06291=1102.506,344.494,-85.854,179.703,17.257,151.749
C06292=1102.511,344.742,-85.887,179.706,17.260,151.749
C06293=1102.517,344.989,-85.921,179.709,17.264,151.749
C06294=1102.523,345.237,-85.955,179.713,17.266,151.749
C06295=1102.529,345.485,-85.989,179.715,17.269,151.749
C06296=1102.533,345.733,-86.023,179.718,17.272,151.749
C06297=1102.539,345.981,-86.056,179.722,17.275,151.749
C06298=1102.545,346.228,-86.090,179.725,17.278,151.749
C06299=1102.551,346.475,-86.124,179.728,17.281,151.749
C06300=1102.556,346.723,-86.157,179.731,17.284,151.750
C06301=1102.562,346.970,-86.191,179.734,17.287,151.750
C06302=1102.568,347.218,-86.225,179.737,17.290,151.750
C06303=1102.574,347.466,-86.259,179.741,17.293,151.750
C06304=1102.578,347.714,-86.293,179.744,17.296,151.750
C06305=1102.584,347.961,-86.327,179.747,17.299,151.750
C06306=1102.590,348.208,-86.361,179.750,17.303,151.750
C06307=1102.596,348.457,-86.395,179.753,17.306,151.750
C06308=1102.602,348.704,-86.429,179.757,17.309,151.751
C06309=1102.607,348.952,-86.463,179.759,17.312,151.751
C06310=1102.613,349.200,-86.497,179.762,17.315,151.751
C06311=1102.619,349.447,-86.531,179.766,17.319,151.751
C06312=1102.625,349.694,-86.565,179.769,17.321,151.751
C06313=1102.630,349.942,-86.599,179.772,17.324,151.751
C06314=1102.635,350.190,-86.633,179.775,17.328,151.751
C06315=1102.642,350.438,-86.667,179.778,17.331,151.752
C06316=1102.648,350.685,-86.701,179.781,17.334,151.752
C06317=1102.653,350.933,-86.736,179.785,17.337,151.752
C06318=1102.659,351.180,-86.770,179.787,17.340,151.752
C06319=1102.664,351.428,-86.803,179.791,17.344,151.752
C06320=1102.670,351.675,-86.837,179.794,17.347,151.752
C06321=1102.676,351.923,-86.872,179.796,17.350,151.753
C06322=1102.682,352.171,-86.906,179.800,17.353,151.753
C06323=1102.687,352.418,-86.940,179.803,17.356,151.753
C06324=1102.693,352.666,-86.975,179.806,17.360,151.753
C06325=1102.698,352.913,-87.009,179.809,17.363,151.753
C06326=1102.705,353.161,-87.043,179.812,17.366,151.753
C06327=1102.710,353.408,-87.078,179.815,17.370,151.754
C06328=1102.716,353.656,-87.112,179.818,17.373,151.754
C06329=1102.722,353.903,-87.146,179.822,17.377,151.754
C06330=1102.727,354.151,-87.181,179.824,17.379,151.754
C06331=1102.733,354.399,-87.215,179.828,17.383,151.754
C06332=1102.738,354.646,-87.250,179.831,17.386,151.755
C06333=1102.744,354.894,-87.284,179.833,17.389,151.755
C06334=1102.749,355.141,-87.319,179.837,17.393,151.755
C06335=1102.756,355.389,-87.353,179.840,17.396,151.755
C06336=1102.761,355.637,-87.388,179.843,17.400,151.756
C06337=1102.767,355.884,-87.422,179.846,17.403,151.756
C06338=1102.775,356.257,-87.474,179.850,17.409,151.756
C06339=1102.784,356.630,-87.526,179.855,17.414,151.756
C06340=1102.792,357.003,-87.579,179.859,17.418,151.757
C06341=1102.801,357.376,-87.630,179.864,17.424,151.757
C06342=1102.806,357.623,-87.665,179.868,17.427,151.757
C06343=1102.813,357.871,-87.700,179.870,17.431,151.758
C06344=1102.818,358.119,-87.734,179.874,17.435,151.758
C06345=1102.824,358.366,-87.769,179.876,17.438,151.758
C06346=1102.830,358.614,-87.804,179.880,17.442,151.758
C06347=1102.836,358.861,-87.838,179.882,17.445,151.759
C06348=1102.841,359.109,-87.873,179.886,17.449,151.759
C06349=1102.847,359.356,-87.909,179.888,17.452,151.759
C06350=1102.853,359.604,-87.943,179.892,17.456,151.759
C06351=1102.858,359.851,-87.977,179.894,17.459,151.760
C06352=1102.864,360.099,-88.013,179.898,17.463,151.760
C06353=1102.870,360.346,-88.047,179.900,17.466,151.760
C06354=1102.875,360.593,-88.083,179.904,17.470,151.761
C06355=1102.882,360.841,-88.117,179.906,17.473,151.761
C06356=1102.887,361.089,-88.152,179.910,17.477,151.761
C06357=1102.892,361.336,-88.187,179.912,17.480,151.761
C06358=1102.898,361.584,-88.222,179.916,17.484,151.762
C06359=1102.904,361.831,-88.257,179.918,17.488,151.762
C06360=1102.909,362.078,-88.291,179.922,17.492,151.762
C06361=1102.915,362.326,-88.327,179.924,17.495,151.763
C06362=1102.920,362.574,-88.362,179.927,17.499,151.763
C06363=1102.927,362.821,-88.397,179.931,17.503,151.763
C06364=1102.932,363.068,-88.432,179.933,17.506,151.764
C06365=1102.938,363.316,-88.467,179.936,17.510,151.764
C06366=1102.944,363.563,-88.503,179.939,17.514,151.764
C06367=1102.949,363.811,-88.537,179.942,17.518,151.765
C06368=1102.955,364.058,-88.572,179.945,17.521,151.765
C06369=1102.961,364.305,-88.608,179.948,17.525,151.765
C06370=1102.966,364.553,-88.642,179.951,17.529,151.766
C06371=1102.972,364.800,-88.678,179.954,17.533,151.766
C06372=1102.978,365.047,-88.713,179.957,17.537,151.766
C06373=1102.984,365.295,-88.748,179.960,17.540,151.767
C06374=1102.989,365.542,-88.783,179.963,17.544,151.767
C06375=1102.995,365.790,-88.819,179.966,17.548,151.767
C06376=1103.001,366.037,-88.854,179.969,17.552,151.768
C06377=1103.007,366.285,-88.889,179.972,17.556,151.768
C06378=1103.012,366.532,-88.925,179.974,17.560,151.769
C06379=1103.017,366.779,-88.960,179.978,17.563,151.769
C06380=1103.023,367.027,-88.996,179.981,17.568,151.769
C06381=1103.029,367.274,-89.031,179.983,17.572,151.770
C06382=1103.035,367.522,-89.067,179.986,17.575,151.770
C06383=1103.040,367.769,-89.102,179.989,17.579,151.771
C06384=1103.046,368.017,-89.137,179.992,17.583,151.771
C06385=1103.051,368.264,-89.173,179.995,17.587,151.771
C06386=1103.058,368.512,-89.208,179.997,17.591,151.772
C06387=1103.063,368.758,-89.244,-180.000,17.595,151.772
C06388=1103.068,369.005,-89.279,-179.996,17.599,151.773
C06389=1103.074,369.253,-89.315,-179.994,17.603,151.773
C06390=1103.082,369.591,-89.363,-179.990,17.609,151.774
C06391=1103.090,369.930,-89.412,-179.986,17.615,151.774
C06392=1103.098,370.268,-89.461,-179.982,17.620,151.775
C06393=1103.106,370.607,-89.510,-179.978,17.626,151.776
C06394=1103.112,370.854,-89.545,-179.975,17.630,151.776
C06395=1103.118,371.101,-89.581,-179.973,17.634,151.776
C06396=1103.123,371.348,-89.616,-179.969,17.638,151.777
C06397=1103.128,371.596,-89.653,-179.966,17.642,151.777
C06398=1103.134,371.843,-89.688,-179.964,17.646,151.778
C06399=1103.140,372.091,-89.724,-179.961,17.650,151.778
C06400=1103.145,372.338,-89.759,-179.958,17.655,151.779
C06401=1103.152,372.585,-89.796,-179.956,17.658,151.779
C06402=1103.158,372.833,-89.831,-179.953,17.663,151.780
C06403=1103.163,373.080,-89.867,-179.949,17.667,151.780
C06404=1103.169,373.327,-89.903,-179.947,17.672,151.781
C06405=1103.174,373.574,-89.939,-179.944,17.675,151.781
C06406=1103.180,373.822,-89.975,-179.941,17.680,151.782
C06407=1103.186,374.069,-90.011,-179.938,17.684,151.782
C06408=1103.192,374.316,-90.046,-179.935,17.688,151.782
C06409=1103.198,374.563,-90.082,-179.933,17.693,151.783
C06410=1103.203,374.811,-90.119,-179.930,17.697,151.784
C06411=1103.209,375.058,-90.154,-179.927,17.701,151.784
C06412=1103.215,375.305,-90.191,-179.924,17.706,151.785
C06413=1103.220,375.553,-90.227,-179.922,17.710,151.785
C06414=1103.226,375.800,-90.262,-179.919,17.714,151.786
C06415=1103.231,376.047,-90.298,-179.916,17.719,151.786
C06416=1103.237,376.295,-90.335,-179.913,17.723,151.787
C06417=1103.243,376.542,-90.371,-179.911,17.727,151.787
C06418=1103.248,376.789,-90.407,-179.908,17.732,151.788
C06419=1103.254,377.036,-90.444,-179.905,17.737,151.789
C06420=1103.260,377.284,-90.479,-179.902,17.741,151.789
C06421=1103.265,377.530,-90.516,-179.899,17.746,151.790
C06422=1103.271,377.778,-90.552,-179.897,17.750,151.790
C06423=1103.277,378.025,-90.588,-179.894,17.754,151.791
C06424=1103.282,378.272,-90.624,-179.891,17.759,151.791
C06425=1103.288,378.519,-90.661,-179.889,17.764,151.792
C06426=1103.295,378.816,-90.704,-179.885,17.769,151.793
C06427=1103.302,379.113,-90.747,-179.882,17.774,151.793
C06428=1103.309,379.410,-90.791,-179.879,17.780,151.794
C06429=1103.315,379.707,-90.835,-179.876,17.785,151.795
C06430=1103.321,379.954,-90.871,-179.873,17.790,151.795
C06431=1103.328,380.201,-90.908,-179.870,17.795,151.796
C06432=1103.332,380.448,-90.944,-179.867,17.799,151.797
C06433=1103.339,380.695,-90.980,-179.865,17.803,151.797
C06434=1103.344,380.943,-91.017,-179.862,17.808,151.798
C06435=1103.350,381.189,-91.053,-179.859,17.813,151.798
C06436=1103.355,381.437,-91.090,-179.857,17.818,151.799
C06437=1103.362,381.684,-91.126,-179.854,17.822,151.800
C06438=1103.367,381.931,-91.163,-179.851,17.827,151.800
C06439=1103.374,382.178,-91.200,-179.848,17.832,151.801
C06440=1103.378,382.426,-91.236,-179.846,17.836,151.802
C06441=1103.385,382.673,-91.272,-179.844,17.841,151.802
C06442=1103.394,383.088,-91.334,-179.838,17.850,151.803
C06443=1103.404,383.502,-91.396,-179.834,17.858,151.805
C06444=1103.413,383.918,-91.457,-179.830,17.866,151.806
C06445=1103.422,384.332,-91.519,-179.826,17.874,151.807
C06446=1103.429,384.579,-91.555,-179.823,17.878,151.808
C06447=1103.434,384.826,-91.592,-179.820,17.884,151.808
C06448=1103.440,385.074,-91.629,-179.818,17.889,151.809
C06449=1103.445,385.320,-91.666,-179.815,17.893,151.810
C06450=1103.451,385.567,-91.703,-179.813,17.899,151.810
C06451=1103.457,385.815,-91.740,-179.810,17.904,151.811
C06452=1103.462,386.062,-91.777,-179.807,17.908,151.812
C06453=1103.468,386.310,-91.814,-179.805,17.913,151.813
C06454=1103.474,386.556,-91.850,-179.802,17.919,151.813
C06455=1103.479,386.803,-91.887,-179.799,17.924,151.814
C06456=1103.485,387.050,-91.925,-179.797,17.929,151.815
C06457=1103.491,387.297,-91.962,-179.794,17.934,151.816
C06458=1103.497,387.544,-91.998,-179.791,17.939,151.816
C06459=1103.503,387.792,-92.035,-179.789,17.944,151.817
C06460=1103.508,388.038,-92.072,-179.786,17.949,151.818
C06461=1103.514,388.285,-92.110,-179.784,17.954,151.819
C06462=1103.519,388.533,-92.147,-179.781,17.959,151.819
C06463=1103.525,388.780,-92.184,-179.779,17.964,151.820
C06464=1103.531,389.027,-92.220,-179.776,17.970,151.821
C06465=1103.537,389.274,-92.258,-179.774,17.975,151.822
C06466=1103.543,389.521,-92.295,-179.771,17.980,151.823
C06467=1103.548,389.768,-92.332,-179.769,17.985,151.823
C06468=1103.554,390.015,-92.370,-179.766,17.990,151.824
C06469=1103.560,390.263,-92.407,-179.764,17.995,151.825
C06470=1103.565,390.510,-92.444,-179.761,18.001,151.826
C06471=1103.572,390.756,-92.481,-179.758,18.007,151.827
C06472=1103.577,391.003,-92.518,-179.755,18.012,151.827
C06473=1103.583,391.251,-92.555,-179.753,18.017,151.828
C06474=1103.588,391.497,-92.592,-179.750,18.022,151.829
C06475=1103.594,391.745,-92.629,-179.748,18.028,151.830
C06476=1103.600,391.991,-92.667,-179.746,18.033,151.831
C06477=1103.606,392.239,-92.705,-179.743,18.039,151.832
C06478=1103.612,392.486,-92.742,-179.741,18.044,151.833
C06479=1103.618,392.733,-92.779,-179.738,18.049,151.833
C06480=1103.623,392.979,-92.817,-179.736,18.055,151.834
C06481=1103.629,393.228,-92.854,-179.733,18.060,151.835
C06482=1103.635,393.474,-92.892,-179.731,18.065,151.836
C06483=1103.641,393.722,-92.929,-179.728,18.071,151.837
C06484=1103.647,393.968,-92.967,-179.726,18.077,151.838
C06485=1103.651,394.216,-93.004,-179.723,18.082,151.839
C06486=1103.657,394.463,-93.042,-179.721,18.088,151.840
C06487=1103.663,394.710,-93.080,-179.719,18.093,151.841
C06488=1103.669,394.957,-93.117,-179.716,18.099,151.842
C06489=1103.675,395.204,-93.155,-179.714,18.104,151.843
C06490=1103.681,395.450,-93.192,-179.712,18.110,151.843
C06491=1103.686,395.698,-93.229,-179.709,18.116,151.844
C06492=1103.691,395.945,-93.268,-179.706,18.122,151.845
C06493=1103.697,396.192,-93.306,-179.704,18.127,151.846
C06494=1103.702,396.405,-93.338,-179.703,18.132,151.847
C06495=1103.707,396.619,-93.370,-179.700,18.137,151.848
C06496=1103.713,396.833,-93.403,-179.698,18.142,151.849
C06497=1103.717,397.046,-93.436,-179.696,18.147,151.850
C06498=1103.722,397.260,-93.469,-179.694,18.152,151.851
C06499=1103.727,397.473,-93.501,-179.692,18.157,151.851
C06500=1103.732,397.686,-93.534,-179.690,18.162,151.852
C06501=1103.737,397.899,-93.566,-179.688,18.167,151.853
C06502=1103.743,398.147,-93.605,-179.685,18.173,151.854
C06503=1103.748,398.395,-93.642,-179.683,18.178,151.855
C06504=1103.754,398.641,-93.680,-179.680,18.185,151.856
C06505=1103.759,398.888,-93.718,-179.678,18.191,151.857
C06506=1103.765,399.135,-93.756,-179.676,18.196,151.858
C06507=1103.771,399.382,-93.794,-179.674,18.202,151.859
C06508=1103.777,399.630,-93.832,-179.671,18.209,151.860
C06509=1103.783,399.876,-93.870,-179.669,18.215,151.861
C06510=1103.789,400.123,-93.908,-179.667,18.220,151.862
C06511=1103.794,400.370,-93.946,-179.665,18.226,151.863
C06512=1103.800,400.617,-93.984,-179.662,18.233,151.864
C06513=1103.805,400.864,-94.022,-179.660,18.238,151.865
C06514=1103.812,401.111,-94.060,-179.657,18.244,151.867
C06515=1103.817,401.359,-94.099,-179.655,18.251,151.868
C06516=1103.823,401.605,-94.137,-179.653,18.257,151.869
C06517=1103.828,401.852,-94.175,-179.651,18.263,151.870
C06518=1103.834,402.100,-94.213,-179.648,18.269,151.871
C06519=1103.840,402.347,-94.251,-179.646,18.275,151.872
C06520=1103.845,402.594,-94.289,-179.644,18.282,151.873
C06521=1103.852,402.840,-94.328,-179.641,18.288,151.874
C06522=1103.857,403.087,-94.366,-179.639,18.294,151.875
C06523=1103.863,403.334,-94.405,-179.637,18.300,151.877
C06524=1103.868,403.581,-94.442,-179.634,18.307,151.878
C06525=1103.874,403.828,-94.481,-179.633,18.313,151.879
C06526=1103.880,404.075,-94.520,-179.630,18.319,151.880
C06527=1103.886,404.322,-94.558,-179.628,18.326,151.881
C06528=1103.892,404.569,-94.596,-179.626,18.332,151.882
C06529=1103.897,404.817,-94.634,-179.623,18.339,151.884
C06530=1103.903,405.063,-94.673,-179.621,18.345,151.885
C06531=1103.909,405.310,-94.711,-179.618,18.351,151.886
C06532=1103.914,405.558,-94.750,-179.617,18.358,151.887
C06533=1103.921,405.804,-94.788,-179.615,18.364,151.888
C06534=1103.926,406.051,-94.827,-179.612,18.371,151.890
C06535=1103.932,406.299,-94.865,-179.610,18.377,151.891
C06536=1103.938,406.545,-94.904,-179.608,18.384,151.892
C06537=1103.943,406.792,-94.942,-179.606,18.390,151.893
C06538=1103.949,407.039,-94.982,-179.603,18.397,151.894
C06539=1103.954,407.286,-95.020,-179.601,18.404,151.896
C06540=1103.960,407.533,-95.058,-179.599,18.411,151.897
C06541=1103.966,407.780,-95.097,-179.597,18.417,151.898
C06542=1103.971,408.027,-95.136,-179.594,18.424,151.899
C06543=1103.977,408.273,-95.175,-179.593,18.430,151.901
C06544=1103.983,408.521,-95.213,-179.590,18.438,151.902
C06545=1103.989,408.767,-95.252,-179.588,18.444,151.903
C06546=1103.994,409.014,-95.291,-179.586,18.451,151.905
C06547=1104.000,409.261,-95.330,-179.584,18.458,151.906
C06548=1104.005,409.508,-95.369,-179.582,18.465,151.907
C06549=1104.011,409.756,-95.407,-179.579,18.472,151.909
C06550=1104.016,409.969,-95.441,-179.577,18.478,151.910
C06551=1104.021,410.182,-95.475,-179.576,18.483,151.911
C06552=1104.026,410.395,-95.508,-179.574,18.490,151.912
C06553=1104.031,410.608,-95.542,-179.572,18.496,151.913
C06554=1104.036,410.822,-95.576,-179.570,18.502,151.914
C06555=1104.041,411.036,-95.609,-179.569,18.508,151.916
C06556=1104.046,411.249,-95.643,-179.566,18.514,151.917
C06557=1104.051,411.462,-95.677,-179.565,18.520,151.918
C06558=1104.056,411.710,-95.716,-179.563,18.527,151.919
C06559=1104.062,411.956,-95.755,-179.561,18.534,151.921
C06560=1104.068,412.203,-95.794,-179.558,18.541,151.922
C06561=1104.073,412.450,-95.833,-179.557,18.549,151.924
C06562=1104.079,412.697,-95.873,-179.554,18.556,151.925
C06563=1104.085,412.944,-95.911,-179.552,18.563,151.926
C06564=1104.091,413.191,-95.950,-179.550,18.570,151.928
C06565=1104.096,413.438,-95.989,-179.548,18.577,151.929
C06566=1104.102,413.685,-96.029,-179.546,18.585,151.931
C06567=1104.108,413.931,-96.068,-179.544,18.592,151.932
C06568=1104.114,414.178,-96.107,-179.542,18.599,151.934
C06569=1104.119,414.425,-96.146,-179.540,18.607,151.935
C06570=1104.125,414.672,-96.186,-179.537,18.614,151.936
C06571=1104.131,414.918,-96.225,-179.536,18.621,151.938
C06572=1104.137,415.165,-96.264,-179.534,18.629,151.939
C06573=1104.142,415.412,-96.303,-179.532,18.636,151.941
C06574=1104.148,415.659,-96.343,-179.529,18.644,151.942
C06575=1104.155,415.906,-96.382,-179.527,18.651,151.944
C06576=1104.160,416.153,-96.421,-179.526,18.658,151.945
C06577=1104.166,416.400,-96.461,-179.524,18.666,151.947
C06578=1104.172,416.646,-96.500,-179.521,18.674,151.948
C06579=1104.178,416.893,-96.540,-179.519,18.681,151.950
C06580=1104.183,417.139,-96.579,-179.517,18.689,151.951
C06581=1104.189,417.387,-96.619,-179.515,18.697,151.953
C06582=1104.195,417.634,-96.658,-179.514,18.704,151.955
C06583=1104.200,417.880,-96.698,-179.512,18.712,151.956
C06584=1104.207,418.127,-96.738,-179.510,18.720,151.958
C06585=1104.211,418.373,-96.777,-179.508,18.727,151.959
C06586=1104.217,418.621,-96.817,-179.506,18.735,151.961
C06587=1104.223,418.867,-96.856,-179.504,18.743,151.963
C06588=1104.229,419.113,-96.896,-179.501,18.751,151.964
C06589=1104.235,419.361,-96.936,-179.500,18.759,151.966
C06590=1104.240,419.607,-96.975,-179.498,18.767,151.968
C06591=1104.246,419.854,-97.015,-179.496,18.775,151.969
C06592=1104.251,420.101,-97.055,-179.495,18.783,151.971
C06593=1104.257,420.348,-97.094,-179.493,18.791,151.973
C06594=1104.264,420.594,-97.134,-179.491,18.799,151.974
C06595=1104.268,420.841,-97.174,-179.489,18.807,151.976
C06596=1104.275,421.088,-97.214,-179.487,18.815,151.977
C06597=1104.281,421.335,-97.254,-179.485,18.823,151.979
C06598=1104.286,421.581,-97.294,-179.483,18.831,151.981
C06599=1104.292,421.828,-97.334,-179.481,18.839,151.982
C06600=1104.298,422.074,-97.374,-179.479,18.847,151.984
C06601=1104.304,422.322,-97.414,-179.477,18.855,151.986
C06602=1104.309,422.568,-97.453,-179.475,18.864,151.988
C06603=1104.315,422.815,-97.494,-179.474,18.872,151.989
C06604=1104.321,423.062,-97.534,-179.472,18.880,151.991
C06605=1104.327,423.307,-97.573,-179.469,18.889,151.993
C06606=1104.332,423.528,-97.609,-179.468,18.896,151.995
C06607=1104.337,423.748,-97.645,-179.467,18.904,151.996
C06608=1104.342,423.969,-97.681,-179.464,18.911,151.998
C06609=1104.347,424.189,-97.717,-179.463,18.919,151.999
C06610=1104.352,424.408,-97.753,-179.461,18.927,152.001
C06611=1104.357,424.629,-97.788,-179.460,18.934,152.003
C06612=1104.362,424.849,-97.824,-179.458,18.942,152.004
C06613=1104.367,425.069,-97.860,-179.457,18.949,152.006
C06614=1104.374,425.316,-97.900,-179.455,18.958,152.008
C06615=1104.379,425.562,-97.941,-179.453,18.966,152.010
C06616=1104.384,425.809,-97.981,-179.452,18.975,152.012
C06617=1104.391,426.055,-98.021,-179.449,18.984,152.013
C06618=1104.396,426.302,-98.062,-179.448,18.993,152.015
C06619=1104.402,426.549,-98.102,-179.446,19.002,152.017
C06620=1104.407,426.795,-98.142,-179.445,19.010,152.019
C06621=1104.413,427.042,-98.183,-179.443,19.019,152.021
C06622=1104.419,427.288,-98.223,-179.441,19.028,152.023
C06623=1104.425,427.535,-98.264,-179.439,19.037,152.025
C06624=1104.430,427.781,-98.304,-179.438,19.046,152.027
C06625=1104.436,428.028,-98.344,-179.436,19.055,152.029
C06626=1104.442,428.275,-98.385,-179.435,19.063,152.031
C06627=1104.448,428.521,-98.425,-179.432,19.073,152.033
C06628=1104.454,428.768,-98.466,-179.431,19.082,152.035
C06629=1104.460,429.015,-98.507,-179.429,19.090,152.037
C06630=1104.465,429.261,-98.547,-179.428,19.100,152.039
C06631=1104.471,429.507,-98.588,-179.426,19.109,152.041
C06632=1104.477,429.754,-98.629,-179.424,19.118,152.043
C06633=1104.483,430.001,-98.669,-179.423,19.127,152.045
C06634=1104.488,430.247,-98.710,-179.421,19.137,152.047
C06635=1104.493,430.494,-98.750,-179.419,19.146,152.049
C06636=1104.500,430.740,-98.791,-179.418,19.155,152.051
C06637=1104.506,430.986,-98.832,-179.417,19.164,152.053
C06638=1104.511,431.233,-98.873,-179.415,19.174,152.055
C06639=1104.517,431.480,-98.913,-179.413,19.183,152.057
C06640=1104.523,431.726,-98.955,-179.411,19.193,152.059
C06641=1104.529,431.973,-98.996,-179.410,19.202,152.061
C06642=1104.534,432.220,-99.036,-179.409,19.211,152.063
C06643=1104.540,432.465,-99.077,-179.407,19.222,152.066
C06644=1104.546,432.712,-99.118,-179.405,19.231,152.068
C06645=1104.552,432.959,-99.158,-179.404,19.240,152.070
C06646=1104.558,433.205,-99.200,-179.402,19.250,152.072
C06647=1104.563,433.452,-99.241,-179.401,19.260,152.074
C06648=1104.569,433.698,-99.282,-179.399,19.270,152.076
C06649=1104.575,433.945,-99.323,-179.398,19.279,152.079
C06650=1104.581,434.191,-99.364,-179.396,19.289,152.081
C06651=1104.586,434.438,-99.405,-179.395,19.299,152.083
C06652=1104.592,434.684,-99.446,-179.394,19.309,152.086
C06653=1104.597,434.930,-99.487,-179.392,19.319,152.088
C06654=1104.603,435.176,-99.528,-179.391,19.329,152.090
C06655=1104.609,435.423,-99.569,-179.389,19.339,152.092
C06656=1104.614,435.670,-99.611,-179.388,19.349,152.095
C06657=1104.620,435.916,-99.652,-179.387,19.359,152.097
C06658=1104.626,436.163,-99.693,-179.386,19.369,152.099
C06659=1104.632,436.409,-99.735,-179.384,19.379,152.102
C06660=1104.638,436.655,-99.776,-179.383,19.389,152.104
C06661=1104.643,436.902,-99.817,-179.381,19.399,152.106
C06662=1104.653,437.320,-99.887,-179.379,19.417,152.110
C06663=1104.658,437.528,-99.923,-179.377,19.426,152.112
C06664=1104.663,437.736,-99.958,-179.377,19.434,152.114
C06665=1104.668,437.946,-99.992,-179.375,19.443,152.116
C06666=1104.673,438.154,-100.028,-179.375,19.452,152.118
C06667=1104.677,438.363,-100.062,-179.373,19.461,152.120
C06668=1104.683,438.572,-100.097,-179.373,19.469,152.123
C06669=1104.688,438.818,-100.140,-179.371,19.480,152.125
C06670=1104.694,439.064,-100.181,-179.369,19.491,152.127
C06671=1104.700,439.311,-100.222,-179.369,19.501,152.130
C06672=1104.706,439.557,-100.264,-179.367,19.512,152.132
C06673=1104.712,439.803,-100.305,-179.365,19.523,152.135
C06674=1104.717,440.049,-100.347,-179.365,19.533,152.137
C06675=1104.723,440.296,-100.389,-179.363,19.544,152.140
C06676=1104.729,440.542,-100.430,-179.363,19.554,152.142
C06677=1104.735,440.788,-100.472,-179.361,19.566,152.145
C06678=1104.740,441.035,-100.514,-179.360,19.577,152.148
C06679=1104.747,441.282,-100.556,-179.358,19.588,152.150
C06680=1104.752,441.528,-100.598,-179.358,19.598,152.153
C06681=1104.758,441.774,-100.639,-179.357,19.610,152.155
C06682=1104.764,442.020,-100.681,-179.355,19.621,152.158
C06683=1104.769,442.267,-100.723,-179.355,19.631,152.161
C06684=1104.775,442.513,-100.764,-179.353,19.643,152.163
C06685=1104.781,442.759,-100.806,-179.352,19.654,152.166
C06686=1104.786,443.005,-100.848,-179.351,19.665,152.168
C06687=1104.792,443.251,-100.890,-179.350,19.676,152.171
C06688=1104.797,443.498,-100.932,-179.349,19.688,152.174
C06689=1104.804,443.744,-100.974,-179.348,19.699,152.177
C06690=1104.810,443.991,-101.016,-179.347,19.710,152.179
C06691=1104.815,444.237,-101.058,-179.347,19.721,152.182
C06692=1104.821,444.483,-101.101,-179.346,19.733,152.185
C06693=1104.827,444.729,-101.142,-179.346,19.744,152.188
C06694=1104.832,444.976,-101.184,-179.346,19.755,152.191
C06695=1104.839,445.222,-101.227,-179.345,19.767,152.193
C06696=1104.844,445.468,-101.269,-179.346,19.777,152.196
C06697=1104.849,445.715,-101.311,-179.346,19.789,152.199
C06698=1104.856,445.960,-101.353,-179.347,19.800,152.202
C06699=1104.861,446.207,-101.395,-179.346,19.811,152.205
C06700=1104.868,446.453,-101.438,-179.347,19.822,152.208
C06701=1104.873,446.700,-101.480,-179.348,19.833,152.211
C06702=1104.878,446.946,-101.522,-179.349,19.844,152.214
C06703=1104.884,447.192,-101.564,-179.350,19.855,152.217
C06704=1104.890,447.438,-101.607,-179.351,19.866,152.220
C06705=1104.896,447.685,-101.649,-179.351,19.877,152.223
C06706=1104.901,447.931,-101.692,-179.353,19.888,152.226
C06707=1104.907,448.177,-101.733,-179.354,19.899,152.229
C06708=1104.913,448.423,-101.776,-179.356,19.910,152.232
C06709=1104.919,448.670,-101.818,-179.357,19.922,152.235
C06710=1104.925,448.916,-101.861,-179.358,19.932,152.238
C06711=1104.930,449.162,-101.903,-179.360,19.943,152.241
C06712=1104.936,449.409,-101.946,-179.362,19.954,152.244
C06713=1104.941,449.655,-101.988,-179.364,19.965,152.247
C06714=1104.948,449.901,-102.030,-179.366,19.976,152.250
C06715=1104.953,450.147,-102.073,-179.367,19.987,152.254
C06716=1104.959,450.394,-102.115,-179.369,19.998,152.257
C06717=1104.555,450.386,-102.243,-179.445,20.226,152.328
C06718=1104.549,450.140,-102.200,-179.443,20.215,152.325
C06719=1104.544,449.893,-102.158,-179.441,20.204,152.322
C06720=1104.537,449.647,-102.115,-179.440,20.193,152.319
C06721=1104.532,449.401,-102.073,-179.438,20.182,152.316
C06722=1104.526,449.154,-102.030,-179.436,20.171,152.312
C06723=1104.520,448.908,-101.988,-179.434,20.160,152.309
C06724=1104.514,448.663,-101.945,-179.433,20.150,152.306
C06725=1104.509,448.416,-101.903,-179.432,20.138,152.303
C06726=1104.503,448.170,-101.860,-179.430,20.127,152.300
C06727=1104.498,447.923,-101.818,-179.429,20.116,152.297
C06728=1104.491,447.678,-101.776,-179.428,20.105,152.294
C06729=1104.485,447.431,-101.733,-179.427,20.094,152.291
C06730=1104.480,447.184,-101.691,-179.426,20.082,152.288
C06731=1104.475,446.939,-101.648,-179.425,20.071,152.285
C06732=1104.469,446.692,-101.607,-179.424,20.060,152.282
C06733=1104.463,446.446,-101.563,-179.424,20.049,152.279
C06734=1104.457,446.199,-101.521,-179.423,20.038,152.276
C06735=1104.451,445.954,-101.479,-179.423,20.026,152.273
C06736=1104.446,445.707,-101.437,-179.422,20.015,152.270
C06737=1104.439,445.461,-101.395,-179.423,20.004,152.267
C06738=1104.434,445.214,-101.353,-179.423,19.992,152.265
C06739=1104.429,444.968,-101.310,-179.422,19.982,152.262
C06740=1104.422,444.722,-101.268,-179.423,19.970,152.259
C06741=1104.417,444.476,-101.226,-179.423,19.959,152.256
C06742=1104.410,444.229,-101.184,-179.424,19.947,152.253
C06743=1104.405,443.983,-101.142,-179.424,19.936,152.250
C06744=1104.399,443.737,-101.100,-179.425,19.925,152.248
C06745=1104.394,443.491,-101.057,-179.426,19.914,152.245
C06746=1104.388,443.245,-101.016,-179.427,19.902,152.242
C06747=1104.382,442.998,-100.974,-179.429,19.890,152.240
C06748=1104.376,442.752,-100.931,-179.429,19.880,152.237
C06749=1104.370,442.505,-100.889,-179.431,19.868,152.234
C06750=1104.364,442.259,-100.848,-179.432,19.857,152.232
C06751=1104.359,442.013,-100.806,-179.433,19.846,152.229
C06752=1104.353,441.767,-100.764,-179.434,19.835,152.226
C06753=1104.347,441.521,-100.722,-179.435,19.824,152.224
C06754=1104.342,441.274,-100.680,-179.437,19.812,152.221
C06755=1104.336,441.028,-100.639,-179.437,19.802,152.218
C06756=1104.330,440.782,-100.597,-179.439,19.791,152.216
C06757=1104.325,440.535,-100.555,-179.440,19.779,152.213
C06758=1104.318,440.289,-100.513,-179.442,19.768,152.211
C06759=1104.312,440.042,-100.472,-179.443,19.758,152.208
C06760=1104.307,439.796,-100.430,-179.444,19.747,152.206
C06761=1104.301,439.550,-100.388,-179.445,19.736,152.203
C06762=1104.295,439.303,-100.347,-179.446,19.726,152.201
C06763=1104.289,439.057,-100.305,-179.448,19.715,152.198
C06764=1104.283,438.811,-100.264,-179.449,19.705,152.196
C06765=1104.278,438.564,-100.222,-179.451,19.694,152.193
C06766=1104.268,438.152,-100.153,-179.453,19.676,152.189
C06767=1104.258,437.740,-100.083,-179.455,19.659,152.185
C06768=1104.249,437.328,-100.014,-179.457,19.641,152.181
C06769=1104.239,436.915,-99.944,-179.460,19.624,152.177
C06770=1104.233,436.669,-99.903,-179.462,19.613,152.175
C06771=1104.227,436.422,-99.862,-179.462,19.603,152.172
C06772=1104.221,436.176,-99.820,-179.464,19.593,152.170
C06773=1104.215,435.930,-99.779,-179.465,19.583,152.168
C06774=1104.209,435.684,-99.738,-179.467,19.573,152.166
C06775=1104.204,435.437,-99.696,-179.468,19.563,152.163
C06776=1104.199,435.190,-99.655,-179.470,19.552,152.161
C06777=1104.193,434.944,-99.613,-179.471,19.543,152.159
C06778=1104.187,434.697,-99.573,-179.473,19.532,152.156
C06779=1104.181,434.451,-99.531,-179.474,19.522,152.154
C06780=1104.176,434.205,-99.491,-179.476,19.512,152.152
C06781=1104.170,433.959,-99.449,-179.477,19.502,152.149
C06782=1104.164,433.712,-99.409,-179.478,19.493,152.147
C06783=1104.158,433.466,-99.367,-179.480,19.483,152.145
C06784=1104.153,433.219,-99.326,-179.481,19.473,152.143
C06785=1104.147,432.973,-99.285,-179.484,19.463,152.141
C06786=1104.141,432.726,-99.244,-179.485,19.454,152.138
C06787=1104.135,432.480,-99.203,-179.487,19.444,152.136
C06788=1104.130,432.233,-99.162,-179.488,19.434,152.134
C06789=1104.124,431.987,-99.120,-179.489,19.425,152.132
C06790=1104.118,431.740,-99.080,-179.492,19.415,152.130
C06791=1104.112,431.493,-99.040,-179.493,19.406,152.128
C06792=1104.106,431.248,-98.999,-179.494,19.396,152.126
C06793=1104.101,431.001,-98.958,-179.496,19.387,152.124
C06794=1104.095,430.754,-98.917,-179.498,19.377,152.121
C06795=1104.089,430.507,-98.876,-179.499,19.368,152.119
C06796=1104.083,430.261,-98.835,-179.501,19.358,152.117
C06797=1104.078,430.014,-98.794,-179.503,19.349,152.115
C06798=1104.071,429.768,-98.754,-179.504,19.340,152.113
C06799=1104.066,429.522,-98.714,-179.506,19.330,152.111
C06800=1104.061,429.275,-98.673,-179.508,19.321,152.109
C06801=1104.055,429.029,-98.631,-179.509,19.312,152.107
C06802=1104.048,428.782,-98.591,-179.511,19.303,152.105
C06803=1104.043,428.535,-98.550,-179.513,19.294,152.103
C06804=1104.037,428.289,-98.510,-179.514,19.285,152.101
C06805=1104.031,428.043,-98.470,-179.516,19.276,152.099
C06806=1104.026,427.796,-98.429,-179.518,19.267,152.097
C06807=1104.020,427.549,-98.388,-179.520,19.258,152.095
C06808=1104.014,427.303,-98.348,-179.521,19.249,152.093
C06809=1104.008,427.056,-98.308,-179.523,19.240,152.091
C06810=1104.002,426.809,-98.267,-179.525,19.232,152.089
C06811=1103.997,426.563,-98.227,-179.527,19.222,152.088
C06812=1103.991,426.316,-98.186,-179.529,19.213,152.086
C06813=1103.985,426.070,-98.146,-179.530,19.205,152.084
C06814=1103.979,425.823,-98.105,-179.532,19.196,152.082
C06815=1103.974,425.577,-98.065,-179.534,19.187,152.080
C06816=1103.968,425.330,-98.026,-179.535,19.179,152.078
C06817=1103.962,425.083,-97.985,-179.538,19.170,152.076
C06818=1103.957,424.863,-97.949,-179.539,19.162,152.075
C06819=1103.952,424.642,-97.913,-179.541,19.154,152.073
C06820=1103.947,424.422,-97.877,-179.542,19.147,152.071
C06821=1103.942,424.202,-97.841,-179.544,19.139,152.070
C06822=1103.937,423.981,-97.805,-179.546,19.131,152.068
C06823=1103.932,423.761,-97.770,-179.547,19.124,152.066
C06824=1103.927,423.541,-97.734,-179.549,19.116,152.065
C06825=1103.921,423.321,-97.698,-179.550,19.109,152.063
C06826=1103.916,423.074,-97.657,-179.552,19.100,152.061
C06827=1103.909,422.827,-97.617,-179.554,19.092,152.060
C06828=1103.904,422.580,-97.577,-179.556,19.084,152.058
C06829=1103.898,422.334,-97.537,-179.558,19.075,152.056
C06830=1103.892,422.088,-97.497,-179.561,19.067,152.054
C06831=1103.887,421.840,-97.457,-179.562,19.058,152.053
C06832=1103.881,421.594,-97.417,-179.564,19.050,152.051
C06833=1103.875,421.347,-97.378,-179.566,19.042,152.049
C06834=1103.869,421.100,-97.337,-179.568,19.034,152.047
C06835=1103.864,420.854,-97.298,-179.570,19.025,152.046
C06836=1103.858,420.607,-97.257,-179.572,19.017,152.044
C06837=1103.852,420.360,-97.218,-179.573,19.010,152.042
C06838=1103.846,420.114,-97.178,-179.575,19.002,152.041
C06839=1103.841,419.867,-97.138,-179.577,18.994,152.039
C06840=1103.835,419.619,-97.099,-179.579,18.986,152.037
C06841=1103.829,419.374,-97.059,-179.581,18.978,152.036
C06842=1103.823,419.127,-97.019,-179.583,18.970,152.034
C06843=1103.817,418.880,-96.979,-179.585,18.962,152.032
C06844=1103.812,418.633,-96.940,-179.587,18.954,152.031
C06845=1103.806,418.386,-96.900,-179.589,18.946,152.029
C06846=1103.801,418.140,-96.860,-179.591,18.938,152.028
C06847=1103.795,417.893,-96.820,-179.594,18.930,152.026
C06848=1103.788,417.646,-96.781,-179.596,18.922,152.024
C06849=1103.783,417.399,-96.742,-179.598,18.914,152.023
C06850=1103.778,417.152,-96.702,-179.599,18.907,152.021
C06851=1103.772,416.906,-96.662,-179.601,18.899,152.020
C06852=1103.766,416.659,-96.623,-179.603,18.891,152.018
C06853=1103.760,416.412,-96.584,-179.605,18.884,152.017
C06854=1103.754,416.165,-96.544,-179.608,18.876,152.015
C06855=1103.748,415.918,-96.505,-179.610,18.868,152.014
C06856=1103.743,415.672,-96.466,-179.611,18.861,152.012
C06857=1103.736,415.425,-96.425,-179.614,18.854,152.011
C06858=1103.731,415.179,-96.386,-179.616,18.846,152.009
C06859=1103.725,414.931,-96.346,-179.618,18.838,152.008
C06860=1103.719,414.684,-96.307,-179.620,18.831,152.006
C06861=1103.714,414.438,-96.268,-179.622,18.824,152.005
C06862=1103.708,414.191,-96.228,-179.624,18.816,152.003
C06863=1103.702,413.944,-96.189,-179.626,18.809,152.002
C06864=1103.696,413.697,-96.150,-179.629,18.801,152.000
C06865=1103.691,413.451,-96.111,-179.630,18.795,151.999
C06866=1103.685,413.204,-96.071,-179.632,18.787,151.997
C06867=1103.680,412.956,-96.033,-179.635,18.780,151.996
C06868=1103.674,412.709,-95.994,-179.636,18.773,151.994
C06869=1103.668,412.463,-95.955,-179.639,18.765,151.993
C06870=1103.662,412.216,-95.915,-179.641,18.758,151.992
C06871=1103.656,411.970,-95.877,-179.643,18.751,151.990
C06872=1103.650,411.723,-95.837,-179.645,18.744,151.989
C06873=1103.645,411.475,-95.799,-179.647,18.736,151.987
C06874=1103.639,411.262,-95.765,-179.650,18.730,151.986
C06875=1103.634,411.048,-95.731,-179.651,18.724,151.985
C06876=1103.630,410.835,-95.697,-179.653,18.718,151.984
C06877=1103.625,410.621,-95.663,-179.654,18.712,151.983
C06878=1103.620,410.407,-95.630,-179.656,18.706,151.981
C06879=1103.615,410.193,-95.596,-179.658,18.700,151.980
C06880=1103.610,409.980,-95.562,-179.660,18.694,151.979
C06881=1103.605,409.767,-95.529,-179.662,18.687,151.978
C06882=1103.599,409.519,-95.489,-179.664,18.681,151.977
C06883=1103.594,409.272,-95.451,-179.666,18.674,151.975
C06884=1103.588,409.025,-95.412,-179.669,18.666,151.974
C06885=1103.582,408.779,-95.373,-179.671,18.660,151.973
C06886=1103.577,408.532,-95.334,-179.673,18.653,151.971
C06887=1103.571,408.285,-95.295,-179.675,18.646,151.970
C06888=1103.565,408.038,-95.257,-179.678,18.639,151.969
C06889=1103.559,407.791,-95.218,-179.679,18.633,151.967
C06890=1103.554,407.544,-95.179,-179.682,18.626,151.966
C06891=1103.548,407.297,-95.140,-179.684,18.619,151.965
C06892=1103.542,407.050,-95.102,-179.686,18.612,151.964
C06893=1103.536,406.803,-95.063,-179.688,18.606,151.962
C06894=1103.531,406.556,-95.025,-179.691,18.599,151.961
C06895=1103.525,406.309,-94.985,-179.692,18.592,151.960
C06896=1103.519,406.062,-94.948,-179.695,18.586,151.959
C06897=1103.514,405.815,-94.909,-179.697,18.579,151.957
C06898=1103.508,405.568,-94.870,-179.700,18.572,151.956
C06899=1103.502,405.321,-94.832,-179.702,18.566,151.955
C06900=1103.497,405.075,-94.793,-179.704,18.559,151.954
C06901=1103.491,404.827,-94.754,-179.706,18.553,151.953
C06902=1103.485,404.581,-94.716,-179.709,18.546,151.951
C06903=1103.480,404.333,-94.678,-179.711,18.540,151.950
C06904=1103.473,404.087,-94.639,-179.713,18.534,151.949
C06905=1103.468,403.840,-94.601,-179.716,18.527,151.948
C06906=1103.462,403.593,-94.563,-179.717,18.521,151.947
C06907=1103.456,403.345,-94.524,-179.720,18.514,151.946
C06908=1103.450,403.099,-94.486,-179.722,18.508,151.944
C06909=1103.445,402.852,-94.448,-179.724,18.502,151.943
C06910=1103.440,402.605,-94.409,-179.727,18.495,151.942
C06911=1103.433,402.357,-94.371,-179.729,18.489,151.941
C06912=1103.428,402.110,-94.333,-179.732,18.483,151.940
C06913=1103.422,401.864,-94.295,-179.734,18.477,151.939
C06914=1103.417,401.617,-94.256,-179.736,18.471,151.938
C06915=1103.410,401.370,-94.218,-179.739,18.464,151.936
C06916=1103.404,401.123,-94.180,-179.741,18.458,151.935
C06917=1103.399,400.876,-94.142,-179.743,18.452,151.934
C06918=1103.393,400.629,-94.104,-179.746,18.446,151.933
C06919=1103.388,400.382,-94.066,-179.748,18.439,151.932
C06920=1103.381,400.135,-94.028,-179.750,18.434,151.931
C06921=1103.376,399.888,-93.989,-179.752,18.428,151.930
C06922=1103.370,399.641,-93.951,-179.755,18.421,151.929
C06923=1103.364,399.394,-93.914,-179.757,18.415,151.928
C06924=1103.359,399.147,-93.875,-179.759,18.409,151.927
C06925=1103.353,398.900,-93.837,-179.762,18.404,151.926
C06926=1103.347,398.653,-93.799,-179.764,18.397,151.925
C06927=1103.342,398.405,-93.762,-179.767,18.392,151.924
C06928=1103.336,398.158,-93.724,-179.769,18.386,151.923
C06929=1103.330,397.912,-93.686,-179.771,18.380,151.922
C06930=1103.326,397.698,-93.653,-179.773,18.375,151.921
C06931=1103.320,397.484,-93.620,-179.775,18.370,151.920
C06932=1103.315,397.270,-93.587,-179.777,18.364,151.919
C06933=1103.310,397.057,-93.554,-179.780,18.359,151.918
C06934=1103.306,396.842,-93.522,-179.782,18.354,151.917
C06935=1103.300,396.629,-93.490,-179.784,18.349,151.916
C06936=1103.295,396.416,-93.457,-179.786,18.344,151.916
C06937=1103.291,396.202,-93.424,-179.788,18.339,151.915
C06938=1103.285,395.954,-93.387,-179.791,18.333,151.914
C06939=1103.279,395.708,-93.349,-179.793,18.328,151.913
C06940=1103.273,395.461,-93.311,-179.795,18.322,151.912
C06941=1103.267,395.214,-93.273,-179.797,18.317,151.911
C06942=1103.263,394.966,-93.236,-179.800,18.311,151.910
C06943=1103.257,394.720,-93.198,-179.803,18.305,151.909
C06944=1103.251,394.473,-93.160,-179.805,18.299,151.908
C06945=1103.245,394.225,-93.123,-179.807,18.294,151.907
C06946=1103.239,393.978,-93.085,-179.810,18.288,151.906
C06947=1103.233,393.731,-93.048,-179.812,18.283,151.905
C06948=1103.227,393.484,-93.010,-179.814,18.277,151.904
C06949=1103.221,393.237,-92.972,-179.817,18.272,151.903
C06950=1103.216,392.990,-92.935,-179.819,18.266,151.902
C06951=1103.211,392.743,-92.897,-179.822,18.260,151.902
C06952=1103.205,392.496,-92.860,-179.825,18.255,151.901
C06953=1103.199,392.249,-92.822,-179.827,18.249,151.900
C06954=1103.193,392.001,-92.785,-179.830,18.244,151.899
C06955=1103.188,391.755,-92.748,-179.832,18.239,151.898
C06956=1103.181,391.508,-92.711,-179.835,18.233,151.897
C06957=1103.176,391.260,-92.674,-179.837,18.228,151.896
C06958=1103.170,391.014,-92.636,-179.840,18.223,151.896
C06959=1103.164,390.766,-92.599,-179.842,18.217,151.895
C06960=1103.158,390.519,-92.561,-179.845,18.212,151.894
C06961=1103.153,390.272,-92.524,-179.847,18.207,151.893
C06962=1103.147,390.025,-92.487,-179.850,18.201,151.892
C06963=1103.141,389.778,-92.450,-179.853,18.196,151.892
C06964=1103.135,389.531,-92.413,-179.855,18.190,151.891
C06965=1103.129,389.285,-92.376,-179.858,18.185,151.890
C06966=1103.124,389.038,-92.339,-179.860,18.180,151.889
C06967=1103.118,388.790,-92.302,-179.863,18.175,151.888
C06968=1103.113,388.543,-92.265,-179.865,18.170,151.887
C06969=1103.107,388.296,-92.227,-179.868,18.165,151.887
C06970=1103.101,388.049,-92.190,-179.871,18.159,151.886
C06971=1103.095,387.802,-92.153,-179.873,18.154,151.885
C06972=1103.089,387.554,-92.116,-179.876,18.149,151.884
C06973=1103.083,387.308,-92.079,-179.878,18.144,151.883
C06974=1103.078,387.061,-92.042,-179.881,18.139,151.883
C06975=1103.073,386.813,-92.005,-179.883,18.134,151.882
C06976=1103.066,386.566,-91.968,-179.886,18.128,151.881
C06977=1103.061,386.319,-91.931,-179.889,18.123,151.880
C06978=1103.055,386.072,-91.894,-179.891,18.118,151.880
C06979=1103.050,385.824,-91.857,-179.894,18.114,151.879
C06980=1103.044,385.578,-91.821,-179.897,18.108,151.878
C06981=1103.038,385.331,-91.784,-179.899,18.103,151.877
C06982=1103.033,385.083,-91.747,-179.902,18.098,151.877
C06983=1103.027,384.836,-91.710,-179.904,18.093,151.876
C06984=1103.021,384.589,-91.674,-179.907,18.088,151.875
C06985=1103.016,384.342,-91.637,-179.910,18.083,151.875
C06986=1103.006,383.927,-91.575,-179.914,18.075,151.873
C06987=1102.997,383.512,-91.513,-179.918,18.067,151.872
C06988=1102.987,383.096,-91.451,-179.923,18.058,151.871
C06989=1102.977,382.682,-91.389,-179.928,18.050,151.870
C06990=1102.972,382.434,-91.353,-179.930,18.045,151.869
C06991=1102.966,382.187,-91.317,-179.933,18.041,151.868
C06992=1102.960,381.940,-91.280,-179.936,18.036,151.868
C06993=1102.954,381.693,-91.244,-179.938,18.031,151.867
C06994=1102.948,381.445,-91.207,-179.941,18.027,151.866
C06995=1102.943,381.199,-91.170,-179.943,18.022,151.866
C06996=1102.937,380.951,-91.134,-179.946,18.017,151.865
C06997=1102.931,380.704,-91.098,-179.949,18.013,151.865
C06998=1102.925,380.457,-91.061,-179.952,18.007,151.864
C06999=1102.920,380.210,-91.025,-179.955,18.003,151.863
C07000=1102.914,379.962,-90.988,-179.957,17.998,151.863
C07001=1102.908,379.715,-90.952,-179.960,17.993,151.862
C07002=1102.902,379.468,-90.915,-179.962,17.989,151.861
C07003=1102.897,379.221,-90.879,-179.965,17.985,151.861
C07004=1102.891,378.974,-90.843,-179.968,17.980,151.860
C07005=1102.885,378.726,-90.806,-179.971,17.975,151.860
C07006=1102.880,378.480,-90.771,-179.974,17.970,151.859
C07007=1102.874,378.232,-90.733,-179.977,17.966,151.858
C07008=1102.868,377.984,-90.698,-179.979,17.962,151.858
C07009=1102.863,377.738,-90.661,-179.981,17.957,151.857
C07010=1102.857,377.490,-90.625,-179.985,17.953,151.857
C07011=1102.851,377.243,-90.589,-179.987,17.948,151.856
C07012=1102.846,376.996,-90.553,-179.990,17.943,151.856
C07013=1102.840,376.749,-90.517,-179.993,17.938,151.855
C07014=1102.834,376.501,-90.481,-179.995,17.934,151.854
C07015=1102.829,376.254,-90.444,-179.998,17.930,151.854
C07016=1102.823,376.007,-90.408,179.999,17.925,151.853
C07017=1102.818,375.760,-90.372,179.996,17.921,151.853
C07018=1102.812,375.512,-90.336,179.993,17.916,151.852
C07019=1102.806,375.265,-90.300,179.991,17.912,151.852
C07020=1102.801,375.018,-90.264,179.988,17.907,151.851
C07021=1102.795,374.770,-90.228,179.985,17.903,151.851
C07022=1102.789,374.523,-90.192,179.982,17.898,151.850
C07023=1102.783,374.276,-90.155,179.980,17.895,151.849
C07024=1102.777,374.028,-90.120,179.977,17.890,151.849
C07025=1102.772,373.781,-90.084,179.974,17.886,151.848
C07026=1102.766,373.534,-90.048,179.971,17.881,151.848
C07027=1102.760,373.287,-90.012,179.969,17.877,151.847
C07028=1102.754,373.040,-89.977,179.965,17.873,151.847
C07029=1102.748,372.792,-89.941,179.962,17.869,151.846
C07030=1102.743,372.545,-89.904,179.959,17.864,151.846
C07031=1102.737,372.298,-89.869,179.957,17.861,151.845
C07032=1102.731,372.050,-89.833,179.954,17.856,151.845
C07033=1102.726,371.803,-89.798,179.951,17.852,151.844
C07034=1102.720,371.555,-89.762,179.949,17.848,151.844
C07035=1102.714,371.308,-89.726,179.946,17.844,151.844
C07036=1102.708,371.061,-89.690,179.942,17.839,151.843
C07037=1102.702,370.814,-89.655,179.939,17.835,151.843
C07038=1102.694,370.425,-89.598,179.935,17.829,151.842
C07039=1102.685,370.037,-89.543,179.931,17.822,151.841
C07040=1102.676,369.649,-89.487,179.926,17.816,151.840
C07041=1102.667,369.261,-89.431,179.922,17.809,151.840
C07042=1102.662,369.013,-89.395,179.919,17.805,151.839
C07043=1102.656,368.766,-89.360,179.916,17.801,151.839
C07044=1102.650,368.518,-89.324,179.913,17.797,151.838
C07045=1102.645,368.271,-89.289,179.910,17.793,151.838
C07046=1102.639,368.024,-89.253,179.907,17.789,151.838
C07047=1102.633,367.777,-89.217,179.904,17.785,151.837
C07048=1102.627,367.529,-89.182,179.901,17.781,151.837
C07049=1102.622,367.282,-89.146,179.899,17.777,151.836
C07050=1102.616,367.034,-89.111,179.896,17.773,151.836
C07051=1102.611,366.787,-89.076,179.892,17.769,151.835
C07052=1102.605,366.540,-89.041,179.890,17.765,151.835
C07053=1102.599,366.292,-89.005,179.887,17.761,151.835
C07054=1102.594,366.045,-88.969,179.884,17.757,151.834
C07055=1102.588,365.797,-88.934,179.881,17.753,151.834
C07056=1102.582,365.550,-88.900,179.878,17.749,151.834
C07057=1102.576,365.302,-88.864,179.876,17.746,151.833
C07058=1102.570,365.055,-88.829,179.872,17.742,151.833
C07059=1102.565,364.807,-88.794,179.869,17.737,151.832
C07060=1102.559,364.560,-88.758,179.867,17.734,151.832
C07061=1102.554,364.313,-88.723,179.863,17.730,151.832
C07062=1102.547,364.065,-88.688,179.861,17.726,151.831
C07063=1102.542,363.818,-88.653,179.858,17.722,151.831
C07064=1102.536,363.571,-88.617,179.854,17.718,151.831
C07065=1102.531,363.323,-88.583,179.852,17.715,151.830
C07066=1102.525,363.075,-88.547,179.848,17.711,151.830
C07067=1102.519,362.828,-88.513,179.846,17.707,151.829
C07068=1102.513,362.581,-88.478,179.843,17.703,151.829
C07069=1102.507,362.333,-88.442,179.840,17.700,151.829
C07070=1102.502,362.086,-88.407,179.837,17.696,151.829
C07071=1102.496,361.839,-88.372,179.833,17.692,151.828
C07072=1102.490,361.591,-88.337,179.831,17.688,151.828
C07073=1102.485,361.344,-88.302,179.828,17.685,151.828
C07074=1102.478,361.096,-88.268,179.825,17.681,151.827
C07075=1102.473,360.849,-88.232,179.822,17.677,151.827
C07076=1102.468,360.601,-88.198,179.819,17.674,151.827
C07077=1102.462,360.353,-88.163,179.816,17.670,151.826
C07078=1102.456,360.106,-88.128,179.813,17.667,151.826
C07079=1102.451,359.859,-88.093,179.810,17.663,151.826
C07080=1102.444,359.611,-88.058,179.807,17.660,151.825
C07081=1102.439,359.364,-88.023,179.804,17.656,151.825
C07082=1102.434,359.116,-87.989,179.801,17.652,151.825
C07083=1102.427,358.869,-87.954,179.798,17.649,151.825
C07084=1102.422,358.621,-87.919,179.795,17.645,151.824
C07085=1102.416,358.374,-87.885,179.792,17.641,151.824
C07086=1102.410,358.126,-87.849,179.789,17.637,151.824
C07087=1102.405,357.879,-87.815,179.786,17.634,151.824
C07088=1102.399,357.631,-87.780,179.782,17.631,151.823
C07089=1102.394,357.384,-87.746,179.780,17.627,151.823
C07090=1102.384,357.010,-87.693,179.775,17.622,151.822
C07091=1102.376,356.637,-87.641,179.770,17.617,151.822
C07092=1102.367,356.263,-87.589,179.766,17.612,151.822
C07093=1102.359,355.890,-87.537,179.761,17.606,151.821
C07094=1102.353,355.643,-87.503,179.758,17.603,151.821
C07095=1102.348,355.395,-87.468,179.756,17.599,151.821
C07096=1102.342,355.148,-87.434,179.752,17.596,151.821
C07097=1102.336,354.900,-87.399,179.749,17.592,151.820
C07098=1102.330,354.653,-87.364,179.747,17.589,151.820
C07099=1102.325,354.405,-87.330,179.743,17.586,151.820
C07100=1102.319,354.158,-87.296,179.740,17.582,151.820
C07101=1102.314,353.910,-87.261,179.737,17.579,151.820
C07102=1102.307,353.662,-87.227,179.734,17.575,151.819
C07103=1102.302,353.415,-87.192,179.731,17.572,151.819
C07104=1102.296,353.168,-87.158,179.728,17.569,151.819
C07105=1102.291,352.920,-87.124,179.724,17.565,151.819
C07106=1102.285,352.672,-87.089,179.722,17.562,151.819
C07107=1102.279,352.424,-87.055,179.719,17.559,151.818
C07108=1102.273,352.177,-87.021,179.715,17.555,151.818
C07109=1102.268,351.929,-86.987,179.713,17.552,151.818
C07110=1102.262,351.682,-86.953,179.709,17.549,151.818
C07111=1102.256,351.434,-86.918,179.706,17.546,151.818
C07112=1102.250,351.187,-86.884,179.703,17.542,151.817
C07113=1102.245,350.939,-86.850,179.700,17.539,151.817
C07114=1102.239,350.692,-86.815,179.697,17.536,151.817
C07115=1102.234,350.444,-86.782,179.694,17.533,151.817
C07116=1102.228,350.196,-86.747,179.691,17.530,151.817
C07117=1102.223,349.949,-86.713,179.687,17.526,151.816
C07118=1102.216,349.701,-86.679,179.684,17.523,151.816
C07119=1102.211,349.453,-86.646,179.682,17.520,151.816
C07120=1102.205,349.205,-86.611,179.678,17.516,151.816
C07121=1102.200,348.958,-86.577,179.675,17.513,151.816
C07122=1102.194,348.710,-86.544,179.672,17.511,151.816
C07123=1102.188,348.463,-86.510,179.669,17.507,151.816
C07124=1102.182,348.216,-86.476,179.666,17.504,151.815
C07125=1102.178,347.968,-86.442,179.662,17.500,151.815
C07126=1102.171,347.720,-86.407,179.660,17.497,151.815
C07127=1102.165,347.472,-86.373,179.657,17.494,151.815
C07128=1102.160,347.224,-86.340,179.653,17.491,151.815
C07129=1102.154,346.977,-86.306,179.650,17.488,151.815
C07130=1102.148,346.729,-86.272,179.647,17.485,151.814
C07131=1102.142,346.482,-86.238,179.644,17.482,151.814
C07132=1102.137,346.234,-86.204,179.641,17.479,151.814
C07133=1102.132,345.986,-86.170,179.638,17.476,151.814
C07134=1102.126,345.739,-86.136,179.634,17.473,151.814
C07135=1102.120,345.491,-86.103,179.631,17.470,151.814
C07136=1102.114,345.244,-86.069,179.628,17.467,151.814
C07137=1102.109,344.996,-86.036,179.625,17.463,151.814
C07138=1102.103,344.748,-86.002,179.622,17.461,151.814
C07139=1102.097,344.501,-85.968,179.619,17.458,151.814
C07140=1102.092,344.253,-85.935,179.615,17.455,151.813
C07141=1102.086,344.006,-85.901,179.612,17.452,151.813
C07142=1102.077,343.634,-85.850,179.608,17.448,151.813
C07143=1102.069,343.263,-85.800,179.603,17.443,151.813
C07144=1102.060,342.892,-85.750,179.598,17.439,151.813
C07145=1102.052,342.521,-85.700,179.593,17.434,151.813
C07146=1102.046,342.273,-85.666,179.590,17.431,151.813
C07147=1102.041,342.025,-85.633,179.587,17.429,151.813
C07148=1102.035,341.778,-85.599,179.583,17.425,151.813
C07149=1102.029,341.530,-85.566,179.581,17.422,151.812
C07150=1102.024,341.282,-85.532,179.577,17.420,151.812
C07151=1102.018,341.034,-85.499,179.575,17.417,151.812
C07152=1102.012,340.786,-85.466,179.571,17.414,151.812
C07153=1102.006,340.539,-85.432,179.568,17.411,151.812
C07154=1102.000,340.292,-85.399,179.565,17.408,151.812
C07155=1101.995,340.044,-85.365,179.561,17.405,151.812
C07156=1101.989,339.796,-85.332,179.558,17.402,151.812
C07157=1101.984,339.548,-85.299,179.555,17.399,151.812
C07158=1101.978,339.300,-85.265,179.552,17.397,151.812
C07159=1101.973,339.052,-85.232,179.548,17.393,151.812
C07160=1101.966,338.805,-85.199,179.545,17.391,151.812
C07161=1101.960,338.557,-85.165,179.542,17.388,151.812
C07162=1101.955,338.309,-85.132,179.539,17.386,151.812
C07163=1101.950,338.062,-85.099,179.536,17.383,151.812
C07164=1101.944,337.814,-85.066,179.532,17.380,151.812
C07165=1101.938,337.566,-85.033,179.529,17.377,151.812
C07166=1101.932,337.319,-85.000,179.526,17.375,151.812
C07167=1101.927,337.071,-84.966,179.523,17.372,151.812
C07168=1101.921,336.823,-84.933,179.519,17.369,151.812
C07169=1101.915,336.575,-84.900,179.516,17.366,151.812
C07170=1101.910,336.327,-84.867,179.513,17.364,151.812
C07171=1101.903,336.080,-84.834,179.510,17.361,151.811
C07172=1101.898,335.831,-84.801,179.507,17.358,151.812
C07173=1101.893,335.584,-84.768,179.503,17.355,151.812
C07174=1101.887,335.336,-84.736,179.500,17.353,151.812
C07175=1101.881,335.088,-84.702,179.497,17.350,151.812
C07176=1101.876,334.841,-84.669,179.494,17.347,151.811
C07177=1101.869,334.593,-84.636,179.491,17.345,151.811
C07178=1101.864,334.345,-84.603,179.487,17.342,151.811
C07179=1101.858,334.098,-84.571,179.484,17.339,151.812
C07180=1101.853,333.850,-84.538,179.481,17.337,151.812
C07181=1101.847,333.602,-84.505,179.478,17.334,151.812
C07182=1101.841,333.354,-84.472,179.475,17.332,151.812
C07183=1101.835,333.106,-84.438,179.472,17.329,151.811
C07184=1101.830,332.859,-84.407,179.468,17.326,151.811
C07185=1101.825,332.611,-84.373,179.465,17.323,151.812
C07186=1101.819,332.363,-84.340,179.462,17.321,151.812
C07187=1101.813,332.115,-84.308,179.458,17.318,151.812
C07188=1101.807,331.867,-84.275,179.455,17.316,151.812
C07189=1101.801,331.619,-84.242,179.452,17.314,151.812
C07190=1101.796,331.372,-84.210,179.448,17.311,151.812
C07191=1101.790,331.124,-84.177,179.445,17.308,151.812
C07192=1101.784,330.876,-84.144,179.442,17.306,151.812
C07193=1101.778,330.628,-84.112,179.439,17.303,151.812
C07194=1101.770,330.251,-84.062,179.434,17.300,151.812
C07195=1101.761,329.873,-84.013,179.429,17.296,151.812
C07196=1101.752,329.496,-83.963,179.423,17.292,151.812
C07197=1101.743,329.119,-83.913,179.418,17.289,151.812
C07198=1101.737,328.872,-83.881,179.415,17.286,151.812
C07199=1101.731,328.624,-83.849,179.412,17.284,151.812
C07200=1101.726,328.375,-83.816,179.409,17.281,151.812
C07201=1101.720,328.128,-83.784,179.406,17.279,151.813
C07202=1101.714,327.880,-83.752,179.403,17.277,151.813
C07203=1101.709,327.632,-83.719,179.399,17.273,151.813
C07204=1101.703,327.384,-83.687,179.395,17.271,151.813
C07205=1101.697,327.136,-83.654,179.392,17.269,151.813
C07206=1101.692,326.889,-83.622,179.389,17.266,151.813
C07207=1101.686,326.640,-83.590,179.386,17.264,151.813
C07208=1101.680,326.393,-83.557,179.382,17.262,151.813
C07209=1101.674,326.145,-83.525,179.379,17.259,151.813
C07210=1101.669,325.897,-83.493,179.376,17.257,151.813
C07211=1101.663,325.649,-83.460,179.373,17.255,151.813
C07212=1101.657,325.402,-83.428,179.370,17.252,151.813
C07213=1101.651,325.153,-83.396,179.366,17.250,151.814
C07214=1101.645,324.906,-83.363,179.363,17.248,151.814
C07215=1101.640,324.658,-83.331,179.360,17.246,151.814
C07216=1101.634,324.410,-83.299,179.356,17.243,151.814
C07217=1101.628,324.162,-83.267,179.353,17.240,151.814
C07218=1101.623,323.915,-83.235,179.349,17.238,151.814
C07219=1101.617,323.666,-83.203,179.346,17.236,151.814
C07220=1101.612,323.419,-83.170,179.343,17.234,151.814
C07221=1101.606,323.170,-83.138,179.340,17.231,151.814
C07222=1101.600,322.922,-83.106,179.336,17.229,151.814
C07223=1101.595,322.675,-83.075,179.333,17.227,151.814
C07224=1101.588,322.427,-83.042,179.330,17.224,151.815
C07225=1101.583,322.180,-83.010,179.326,17.222,151.815
C07226=1101.578,321.931,-82.978,179.323,17.220,151.815
C07227=1101.572,321.684,-82.946,179.320,17.217,151.815
C07228=1101.566,321.435,-82.914,179.317,17.215,151.815
C07229=1101.561,321.188,-82.882,179.313,17.213,151.815
C07230=1101.555,320.940,-82.850,179.310,17.211,151.815
C07231=1101.549,320.691,-82.818,179.307,17.208,151.815
C07232=1101.544,320.444,-82.787,179.303,17.206,151.816
C07233=1101.538,320.196,-82.755,179.300,17.204,151.816
C07234=1101.532,319.948,-82.723,179.297,17.202,151.816
C07235=1101.527,319.700,-82.690,179.293,17.200,151.816
C07236=1101.522,319.452,-82.659,179.290,17.197,151.816
C07237=1101.516,319.204,-82.627,179.287,17.195,151.816
C07238=1101.510,318.956,-82.595,179.284,17.193,151.816
C07239=1101.505,318.709,-82.563,179.280,17.191,151.816
C07240=1101.499,318.461,-82.531,179.277,17.189,151.817
C07241=1101.494,318.212,-82.500,179.274,17.186,151.817
C07242=1101.488,317.964,-82.468,179.270,17.184,151.817
C07243=1101.482,317.717,-82.437,179.267,17.182,151.817
C07244=1101.477,317.469,-82.405,179.264,17.179,151.817
C07245=1101.471,317.221,-82.373,179.260,17.177,151.817
C07246=1101.462,316.836,-82.324,179.256,17.174,151.817
C07247=1101.454,316.453,-82.275,179.250,17.170,151.818
C07248=1101.445,316.068,-82.226,179.245,17.167,151.818
C07249=1101.437,315.683,-82.177,179.240,17.164,151.818
C07250=1101.432,315.436,-82.145,179.236,17.162,151.818
C07251=1101.425,315.188,-82.114,179.233,17.160,151.818
C07252=1101.420,314.940,-82.083,179.230,17.157,151.819
C07253=1101.414,314.691,-82.051,179.226,17.155,151.819
C07254=1101.408,314.444,-82.019,179.223,17.153,151.819
C07255=1101.403,314.196,-81.989,179.219,17.151,151.819
C07256=1101.397,313.948,-81.957,179.216,17.149,151.819
